CASE nPhase OF
	0:
		// 初始 Undefined -> Aborted。
		Composite(Ctrl := Ctrl, Context := Context, ServiceId := 10);
		nPhase := 1;
	1:
		Ctrl.PackMLIn.eCommand := E_PackMLCommand.Clear;
		Ctrl.PackMLIn.bCommandChangeRequest := TRUE;
		Composite(Ctrl := Ctrl, Context := Context, ServiceId := 10);
		nPhase := 2;
	2:
		Ctrl.PackMLIn.bCommandChangeRequest := FALSE;
		Composite(Ctrl := Ctrl, Context := Context, ServiceId := 10);
		nPhase := 3;
	3:
		Ctrl.PackMLIn.eCommand := E_PackMLCommand.Reset;
		Ctrl.PackMLIn.bCommandChangeRequest := TRUE;
		Composite(Ctrl := Ctrl, Context := Context, ServiceId := 10);
		nPhase := 4;
	4:
		Ctrl.PackMLIn.bCommandChangeRequest := FALSE;
		Composite(Ctrl := Ctrl, Context := Context, ServiceId := 10);
		nPhase := 5;
	5:
		// Starting 發現 definition 尚未設定，加入 framework error 並排入 Stop。
		Ctrl.PackMLIn.eCommand := E_PackMLCommand.Start;
		Ctrl.PackMLIn.bCommandChangeRequest := TRUE;
		Composite(Ctrl := Ctrl, Context := Context, ServiceId := 10);
		AssertTrue(
			Condition :=
				Composite.Status.ErrorList[1].MainErrorId =
				TO_UDINT(E_CompositeServiceErrorCode.NotConfigured),
			Message := 'Unconfigured Composite must publish NotConfigured.'
		);
		nPhase := 6;
	6:
		// 下一掃描由 queued Stop 將 Starting 安全帶回 Stopped。
		Composite(Ctrl := Ctrl, Context := Context, ServiceId := 10);
		AssertTrue(
			Condition := Composite.Status.PackMLOut.eStateCurrent = E_PackMLState.Stopped,
			Message := 'Unconfigured Composite must follow the safe Stop path.'
		);
		nPhase := 0;
		TEST_FINISHED();
END_CASE
END_METHOD

END_FUNCTION_BLOCK

// ---- Fakes/FB_TestCompositeService.TcPOU
FUNCTION_BLOCK FB_TestCompositeService EXTENDS FB_CompositeServiceBase
VAR_INPUT
	DependencyOne : UDINT;
	DependencyTwo : UDINT;
	DependencyCount : UINT;
	ExecuteResult : E_PackMLHookResult := E_PackMLHookResult.Busy;
END_VAR

M_UpdateCompositeService();

METHOD PROTECTED H_DeclareServices
IF DependencyCount >= 1 THEN
	M_AddDependency(ServiceId := DependencyOne);
END_IF
IF DependencyCount >= 2 THEN
	M_AddDependency(ServiceId := DependencyTwo);
END_IF
END_METHOD

METHOD PROTECTED H_OnCompositeExecute : E_PackMLHookResult
VAR_INPUT
	bFirstScan : BOOL;
END_VAR
H_OnCompositeExecute := ExecuteResult;
END_METHOD

METHOD PUBLIC M_TestAddDependencyOutsideDefinition : BOOL
VAR_INPUT
	ServiceIdValue : UDINT;
END_VAR
M_TestAddDependencyOutsideDefinition := M_AddDependency(ServiceId := ServiceIdValue);
END_METHOD

METHOD PUBLIC M_TestFailSequence
VAR_INPUT
	FailedServiceId : UDINT;
END_VAR
M_FailSequence(
	ErrorCode := E_CompositeServiceErrorCode.None,
	FailedServiceId := FailedServiceId,
	SourceErrorId := 0,
	Message := 'Test failure'
);
END_METHOD

END_FUNCTION_BLOCK

// ---- POUs/Test Suites/Service/FB_SetMaterialServiceTests.TcPOU
FUNCTION_BLOCK FB_SetMaterialServiceTests EXTENDS TcUnit.FB_TestSuite

ModifyUsesTheStartingSnapshot();
ClearAndClearAllAffectOnlyTheirDocumentedScope();
InvalidTargetStopsWithAStableError();
MissingTargetIsRejected();
DuplicateTargetIsRejected();
UnsupportedCommandIsRejected();

METHOD ClearAndClearAllAffectOnlyTheirDocumentedScope
VAR_INST
	Service : FB_SetMaterialService;
	Ctrl : ST_ServiceCtrl;
	Context : ST_ServiceContext;
	Param : ST_MaterialParam;
	Wafers : ARRAY[1..2] OF ST_WaferStatus;
	nPhase : UINT;
END_VAR
TEST('ClearAndClearAllAffectOnlyTheirDocumentedScope');

CASE nPhase OF
	0:
		Wafers[1].EndpointId := 1;
		Wafers[2].EndpointId := 2;
		Wafers[1].MaterialContext.Id := 'A';
		Wafers[2].MaterialContext.Id := 'B';
		Service(
			Ctrl := Ctrl,
			Context := Context,
			ServiceId := 2,
			Param := Param,
			WaferStatusList := Wafers
		);
		nPhase := 1;
		1: Ctrl.PackMLIn.eCommand := E_PackMLCommand.Clear;
		Ctrl.PackMLIn.bCommandChangeRequest := TRUE;
		Service(
			Ctrl := Ctrl,
			Context := Context,
			ServiceId := 2,
			Param := Param,
			WaferStatusList := Wafers
		);
		nPhase := 2;
		2: Ctrl.PackMLIn.bCommandChangeRequest := FALSE;
		Service(
			Ctrl := Ctrl,
			Context := Context,
			ServiceId := 2,
			Param := Param,
			WaferStatusList := Wafers
		);
		nPhase := 3;
		3: Ctrl.PackMLIn.eCommand := E_PackMLCommand.Reset;
		Ctrl.PackMLIn.bCommandChangeRequest := TRUE;
		Service(
			Ctrl := Ctrl,
			Context := Context,
			ServiceId := 2,
			Param := Param,
			WaferStatusList := Wafers
		);
		nPhase := 4;
		4: Ctrl.PackMLIn.bCommandChangeRequest := FALSE;
		Service(
			Ctrl := Ctrl,
			Context := Context,
			ServiceId := 2,
			Param := Param,
			WaferStatusList := Wafers
		);
		nPhase := 5;
	5:
		Param.CmdType := E_SetMaterialCmdType.Clear;
		Param.TargetEndpointId := 1;
		Ctrl.PackMLIn.eCommand := E_PackMLCommand.Start;
		Ctrl.PackMLIn.bCommandChangeRequest := TRUE;
		Service(
			Ctrl := Ctrl,
			Context := Context,
			ServiceId := 2,
			Param := Param,
			WaferStatusList := Wafers
		);
		nPhase := 6;
	6:
		Service(
			Ctrl := Ctrl,
			Context := Context,
			ServiceId := 2,
			Param := Param,
			WaferStatusList := Wafers
		);
		AssertTrue(
			Condition := (Wafers[1].MaterialContext.Id = '')
				AND (Wafers[2].MaterialContext.Id = 'B'),
			Message := 'Clear must affect only the selected endpoint.'
		);
		nPhase := 7;
	7:
		Ctrl.PackMLIn.bCommandChangeRequest := FALSE;
		Service(
			Ctrl := Ctrl,
			Context := Context,
			ServiceId := 2,
			Param := Param,
			WaferStatusList := Wafers
		);
		nPhase := 8;
	8:
		Ctrl.PackMLIn.eCommand := E_PackMLCommand.Reset;
		Ctrl.PackMLIn.bCommandChangeRequest := TRUE;
		Service(
			Ctrl := Ctrl,
			Context := Context,
			ServiceId := 2,
			Param := Param,
			WaferStatusList := Wafers
		);
		nPhase := 9;
	9:
		Ctrl.PackMLIn.bCommandChangeRequest := FALSE;
		Service(
			Ctrl := Ctrl,
			Context := Context,
			ServiceId := 2,
			Param := Param,
			WaferStatusList := Wafers
		);
		nPhase := 10;
	10:
		Wafers[1].MaterialContext.Id := 'A2';
		Param.CmdType := E_SetMaterialCmdType.ClearAll;
		Param.TargetEndpointId := 0;
		Ctrl.PackMLIn.eCommand := E_PackMLCommand.Start;
		Ctrl.PackMLIn.bCommandChangeRequest := TRUE;
		Service(
			Ctrl := Ctrl,
			Context := Context,
			ServiceId := 2,
			Param := Param,
			WaferStatusList := Wafers
		);
		nPhase := 11;
	11:
		Service(
			Ctrl := Ctrl,
			Context := Context,
			ServiceId := 2,
			Param := Param,
			WaferStatusList := Wafers
		);
		AssertTrue(
			Condition := (Wafers[1].MaterialContext.Id = '')
				AND (Wafers[2].MaterialContext.Id = ''),
			Message := 'ClearAll must clear every material context and ignore TargetEndpointId.'
		);
		nPhase := 0;
		TEST_FINISHED();
END_CASE
END_METHOD

METHOD DuplicateTargetIsRejected
VAR_INST
	Service : FB_SetMaterialService;
	Ctrl : ST_ServiceCtrl;
	Context : ST_ServiceContext;
	Param : ST_MaterialParam;
	Wafers : ARRAY[1..2] OF ST_WaferStatus;
	nPhase : UINT;
END_VAR
TEST('DuplicateTargetIsRejected');

CASE nPhase OF
	0: Wafers[1].EndpointId := 7;
	Wafers[2].EndpointId := 7;
	Service(
		Ctrl := Ctrl,
		Context := Context,
		ServiceId := 5,
		Param := Param,
		WaferStatusList := Wafers
	);
	nPhase := 1;
	1: Ctrl.PackMLIn.eCommand := E_PackMLCommand.Clear;
	Ctrl.PackMLIn.bCommandChangeRequest := TRUE;
	Service(
		Ctrl := Ctrl,
		Context := Context,
		ServiceId := 5,
		Param := Param,
		WaferStatusList := Wafers
	);
	nPhase := 2;
	2: Ctrl.PackMLIn.bCommandChangeRequest := FALSE;
	Service(
		Ctrl := Ctrl,
		Context := Context,
		ServiceId := 5,
		Param := Param,
		WaferStatusList := Wafers
	);
	nPhase := 3;
	3: Ctrl.PackMLIn.eCommand := E_PackMLCommand.Reset;
	Ctrl.PackMLIn.bCommandChangeRequest := TRUE;
	Service(
		Ctrl := Ctrl,
		Context := Context,
		ServiceId := 5,
		Param := Param,
		WaferStatusList := Wafers
	);
	nPhase := 4;
	4: Ctrl.PackMLIn.bCommandChangeRequest := FALSE;
	Service(
		Ctrl := Ctrl,
		Context := Context,
		ServiceId := 5,
		Param := Param,
		WaferStatusList := Wafers
	);
	nPhase := 5;
	5:
		// Arrange：兩個 storage slot 宣告同一個外部 EndpointId。
		Param.CmdType := E_SetMaterialCmdType.Modify;
		Param.TargetEndpointId := 7;
		Ctrl.PackMLIn.eCommand := E_PackMLCommand.Start;
		Ctrl.PackMLIn.bCommandChangeRequest := TRUE;
		// Act
		Service(
			Ctrl := Ctrl,
			Context := Context,
			ServiceId := 5,
			Param := Param,
			WaferStatusList := Wafers
		);
		// Assert
		AssertTrue(
			Condition :=
				Service.Status.ErrorList[1].MainErrorId =
				TO_UDINT(E_FrameworkServiceErrorCode.SetMaterial_DuplicateTaEpId),
			Message := 'Duplicate target identity must be rejected before modifying either wafer.'
		);
		AssertTrue(
			Condition := (Wafers[1].MaterialContext.Id = '')
				AND (Wafers[2].MaterialContext.Id = ''),
			Message := 'Rejected duplicate target must not mutate material state.'
		);
		nPhase := 0;
		TEST_FINISHED();
END_CASE
END_METHOD

METHOD InvalidTargetStopsWithAStableError
VAR_INST
	Service : FB_SetMaterialService;
	Ctrl : ST_ServiceCtrl;
	Context : ST_ServiceContext;
	Param : ST_MaterialParam;
	Wafers : ARRAY[1..2] OF ST_WaferStatus;
	nPhase : UINT;
END_VAR
TEST('InvalidTargetStopsWithAStableError');

CASE nPhase OF
	0:
		Service(
			Ctrl := Ctrl,
			Context := Context,
			ServiceId := 3,
			Param := Param,
			WaferStatusList := Wafers
		);
		nPhase := 1;
		1: Ctrl.PackMLIn.eCommand := E_PackMLCommand.Clear;
		Ctrl.PackMLIn.bCommandChangeRequest := TRUE;
		Service(
			Ctrl := Ctrl,
			Context := Context,
			ServiceId := 3,
			Param := Param,
			WaferStatusList := Wafers
		);
		nPhase := 2;
		2: Ctrl.PackMLIn.bCommandChangeRequest := FALSE;
		Service(
			Ctrl := Ctrl,
			Context := Context,
			ServiceId := 3,
			Param := Param,
			WaferStatusList := Wafers
		);
		nPhase := 3;
		3: Ctrl.PackMLIn.eCommand := E_PackMLCommand.Reset;
		Ctrl.PackMLIn.bCommandChangeRequest := TRUE;
		Service(
			Ctrl := Ctrl,
			Context := Context,
			ServiceId := 3,
			Param := Param,
			WaferStatusList := Wafers
		);
		nPhase := 4;
		4: Ctrl.PackMLIn.bCommandChangeRequest := FALSE;
		Service(
			Ctrl := Ctrl,
			Context := Context,
			ServiceId := 3,
			Param := Param,
			WaferStatusList := Wafers
		);
		nPhase := 5;
	5:
		// Arrange：Modify/Clear 的 TargetEndpointId=0 是明確輸入錯誤。
		Param.CmdType := E_SetMaterialCmdType.Modify;
		Param.TargetEndpointId := 0;
		Ctrl.PackMLIn.eCommand := E_PackMLCommand.Start;
		Ctrl.PackMLIn.bCommandChangeRequest := TRUE;
		Service(
			Ctrl := Ctrl,
			Context := Context,
			ServiceId := 3,
			Param := Param,
			WaferStatusList := Wafers
		);
		AssertTrue(
			Condition :=
				Service.Status.ErrorList[1].MainErrorId =
				TO_UDINT(E_FrameworkServiceErrorCode.SetMaterial_TaEpIdRequired),
			Message := 'Zero target must publish the required-target error.'
		);
		nPhase := 6;
	6:
		Service(
			Ctrl := Ctrl,
			Context := Context,
			ServiceId := 3,
			Param := Param,
			WaferStatusList := Wafers
		);
		AssertTrue(
			Condition := Service.Status.PackMLOut.eStateCurrent = E_PackMLState.Stopped,
			Message := 'Invalid material request must follow the safe Stop path.'
		);
		nPhase := 0;
		TEST_FINISHED();
END_CASE
END_METHOD

METHOD MissingTargetIsRejected
VAR_INST
	Service : FB_SetMaterialService;
	Ctrl : ST_ServiceCtrl;
	Context : ST_ServiceContext;
	Param : ST_MaterialParam;
	Wafers : ARRAY[1..2] OF ST_WaferStatus;
	nPhase : UINT;
END_VAR
TEST('MissingTargetIsRejected');

CASE nPhase OF
	0: Wafers[1].EndpointId := 10;
	Wafers[2].EndpointId := 20;
	Service(
		Ctrl := Ctrl,
		Context := Context,
		ServiceId := 4,
		Param := Param,
		WaferStatusList := Wafers
	);
	nPhase := 1;
	1: Ctrl.PackMLIn.eCommand := E_PackMLCommand.Clear;
	Ctrl.PackMLIn.bCommandChangeRequest := TRUE;
	Service(
		Ctrl := Ctrl,
		Context := Context,
		ServiceId := 4,
		Param := Param,
		WaferStatusList := Wafers
	);
	nPhase := 2;
	2: Ctrl.PackMLIn.bCommandChangeRequest := FALSE;
	Service(
		Ctrl := Ctrl,
		Context := Context,
		ServiceId := 4,
		Param := Param,
		WaferStatusList := Wafers
	);
	nPhase := 3;
	3: Ctrl.PackMLIn.eCommand := E_PackMLCommand.Reset;
	Ctrl.PackMLIn.bCommandChangeRequest := TRUE;
	Service(
		Ctrl := Ctrl,
		Context := Context,
		ServiceId := 4,
		Param := Param,
		WaferStatusList := Wafers
	);
	nPhase := 4;
	4: Ctrl.PackMLIn.bCommandChangeRequest := FALSE;
	Service(
		Ctrl := Ctrl,
		Context := Context,
		ServiceId := 4,
		Param := Param,
		WaferStatusList := Wafers
	);
	nPhase := 5;
	5:
		// Arrange：使用非零但不存在的 EndpointId。
		Param.CmdType := E_SetMaterialCmdType.Clear;
		Param.TargetEndpointId := 99;
		Ctrl.PackMLIn.eCommand := E_PackMLCommand.Start;
		Ctrl.PackMLIn.bCommandChangeRequest := TRUE;
		// Act
		Service(
			Ctrl := Ctrl,
			Context := Context,
			ServiceId := 4,
			Param := Param,
			WaferStatusList := Wafers
		);
		// Assert
		AssertTrue(
			Condition :=
				Service.Status.ErrorList[1].MainErrorId =
				TO_UDINT(E_FrameworkServiceErrorCode.SetMaterial_TaEpNotFound),
			Message := 'Unknown target must publish the not-found error.'
		);
		nPhase := 0;
		TEST_FINISHED();
END_CASE
END_METHOD

METHOD ModifyUsesTheStartingSnapshot
VAR_INST
	Service : FB_SetMaterialService;
	Ctrl : ST_ServiceCtrl;
	Context : ST_ServiceContext;
	Param : ST_MaterialParam;
	Wafers : ARRAY[1..2] OF ST_WaferStatus;
	nPhase : UINT;
END_VAR
TEST('ModifyUsesTheStartingSnapshot');

CASE nPhase OF
	0:
		Wafers[1].EndpointId := 101;
		Wafers[2].EndpointId := 102;
		Service(
			Ctrl := Ctrl,
			Context := Context,
			ServiceId := 1,
			Param := Param,
			WaferStatusList := Wafers
		);
		nPhase := 1;
	1:
		Ctrl.PackMLIn.eCommand := E_PackMLCommand.Clear;
		Ctrl.PackMLIn.bCommandChangeRequest := TRUE;
		Service(
			Ctrl := Ctrl,
			Context := Context,
			ServiceId := 1,
			Param := Param,
			WaferStatusList := Wafers
		);
		nPhase := 2;
	2:
		Ctrl.PackMLIn.bCommandChangeRequest := FALSE;
		Service(
			Ctrl := Ctrl,
			Context := Context,
			ServiceId := 1,
			Param := Param,
			WaferStatusList := Wafers
		);
		nPhase := 3;
	3:
		Ctrl.PackMLIn.eCommand := E_PackMLCommand.Reset;
		Ctrl.PackMLIn.bCommandChangeRequest := TRUE;
		Service(
			Ctrl := Ctrl,
			Context := Context,
			ServiceId := 1,
			Param := Param,
			WaferStatusList := Wafers
		);
		nPhase := 4;
	4:
		Ctrl.PackMLIn.bCommandChangeRequest := FALSE;
		Service(
			Ctrl := Ctrl,
			Context := Context,
			ServiceId := 1,
			Param := Param,
			WaferStatusList := Wafers
		);
		nPhase := 5;
	5:
		// Arrange：Starting 驗證並 snapshot Modify 參數。
		Param.CmdType := E_SetMaterialCmdType.Modify;
		Param.TargetEndpointId := 101;
		Param.MaterialId := 'WAFER-A';
		Param.MaterialOperateState := E_MaterialOperateState.Processing;
		Ctrl.PackMLIn.eCommand := E_PackMLCommand.Start;
		Ctrl.PackMLIn.bCommandChangeRequest := TRUE;
		Service(
			Ctrl := Ctrl,
			Context := Context,
			ServiceId := 1,
			Param := Param,
			WaferStatusList := Wafers
		);
		Param.MaterialId := 'MUTATED-AFTER-START';
		nPhase := 6;
	6:
		// Act：Execute 必須使用 Starting 的 snapshot，而不是目前輸入。
		Service(
			Ctrl := Ctrl,
			Context := Context,
			ServiceId := 1,
			Param := Param,
			WaferStatusList := Wafers
		);
		AssertTrue(
			Condition :=
				(Wafers[1].MaterialContext.Id = 'WAFER-A')
				AND (Wafers[1].MaterialContext.OperationState = E_MaterialOperateState.Processing),
			Message := 'Modify must use the snapshotted material context.'
		);
		AssertTrue(
			Condition := Wafers[2].MaterialContext.Id = '',
			Message := 'Modify must not change another endpoint.'
		);
		nPhase := 0;
		TEST_FINISHED();
END_CASE
END_METHOD

METHOD UnsupportedCommandIsRejected
VAR_INST
	Service : FB_SetMaterialService;
	Ctrl : ST_ServiceCtrl;
	Context : ST_ServiceContext;
	Param : ST_MaterialParam;
	Wafers : ARRAY[1..2] OF ST_WaferStatus;
	nPhase : UINT;
END_VAR
VAR
	nInvalidCommand : INT := 9999;
END_VAR
TEST('UnsupportedCommandIsRejected');

CASE nPhase OF
	0: Wafers[1].EndpointId := 1;
	Service(
		Ctrl := Ctrl,
		Context := Context,
		ServiceId := 6,
		Param := Param,
		WaferStatusList := Wafers
	);
	nPhase := 1;
	1: Ctrl.PackMLIn.eCommand := E_PackMLCommand.Clear;
	Ctrl.PackMLIn.bCommandChangeRequest := TRUE;
	Service(
		Ctrl := Ctrl,
		Context := Context,
		ServiceId := 6,
		Param := Param,
		WaferStatusList := Wafers
	);
	nPhase := 2;
	2: Ctrl.PackMLIn.bCommandChangeRequest := FALSE;
	Service(
		Ctrl := Ctrl,
		Context := Context,
		ServiceId := 6,
		Param := Param,
		WaferStatusList := Wafers
	);
	nPhase := 3;
	3: Ctrl.PackMLIn.eCommand := E_PackMLCommand.Reset;
	Ctrl.PackMLIn.bCommandChangeRequest := TRUE;
	Service(
		Ctrl := Ctrl,
		Context := Context,
		ServiceId := 6,
		Param := Param,
		WaferStatusList := Wafers
	);
	nPhase := 4;
	4: Ctrl.PackMLIn.bCommandChangeRequest := FALSE;
	Service(
		Ctrl := Ctrl,
		Context := Context,
		ServiceId := 6,
		Param := Param,
		WaferStatusList := Wafers
	);
	nPhase := 5;
	5:
		// Arrange：模擬反序列化或上游資料損壞造成的未知 enum 值。
		// 故意繞過 strict enum 的編譯期保護，模擬外部資料或記憶體損壞。
		MEMCPY(
			ADR(Param.CmdType),
			ADR(nInvalidCommand),
			SIZEOF(Param.CmdType));
		Param.TargetEndpointId := 1;
		Ctrl.PackMLIn.eCommand := E_PackMLCommand.Start;
		Ctrl.PackMLIn.bCommandChangeRequest := TRUE;
		// Act
		Service(
			Ctrl := Ctrl,
			Context := Context,
			ServiceId := 6,
			Param := Param,
			WaferStatusList := Wafers
		);
		// Assert
		AssertTrue(
			Condition :=
				Service.Status.ErrorList[1].MainErrorId =
				TO_UDINT(E_FrameworkServiceErrorCode.SetMaterial_InvalidCmd),
			Message := 'Unknown material command must publish the invalid-command error.'
		);
		nPhase := 0;
		TEST_FINISHED();
END_CASE
END_METHOD

END_FUNCTION_BLOCK

// ---- POUs/Test Suites/Service/FB_ServiceCallerTests.TcPOU
FUNCTION_BLOCK FB_ServiceCallerTests EXTENDS TcUnit.FB_TestSuite

UnconfiguredCallerRejectsRequests();
ConfiguredCallerDelegatesAndAdvancesRequestIds();

METHOD UnconfiguredCallerRejectsRequests
VAR_INST
	Caller : FB_ServiceCaller;
	Param : ST_TestServiceParam;
	Snapshot : ST_ServiceExecutionSnapshot;
END_VAR
TEST('UnconfiguredCallerRejectsRequests');

AssertTrue(
	Condition := Caller.M_Start(
		ServiceId := 1,
		Parameters := Param
	) = E_ServiceCallSubmitResult.CallerNotConfigured,
	Message := 'Unconfigured Start must be rejected.'
);
AssertTrue(
	Condition := Caller.M_Command(
		ServiceId := 1,
		Command := E_PackMLCommand.Stop
	) = E_ServiceCallSubmitResult.CallerNotConfigured,
	Message := 'Unconfigured command must be rejected.'
);
AssertFalse(
	Condition := Caller.M_GetServiceSnapshot(ServiceId := 1, Snapshot => Snapshot),
	Message := 'Unconfigured snapshot query must fail.'
);

TEST_FINISHED();
END_METHOD

METHOD ConfiguredCallerDelegatesAndAdvancesRequestIds
VAR_INST
	Caller : FB_ServiceCaller;
	Coordinator : FB_ServiceCoordinator;
	CompositeUpperCtrl : ST_ServiceCtrl;
	CompositeEffectiveCtrl : ST_ServiceCtrl;
	CompositeUpperParam : ST_TestServiceParam;
	CompositeEffectiveParam : ST_TestServiceParam;
	CompositeStatus : ST_ServiceStatus;
	ChildUpperCtrl : ST_ServiceCtrl;
	ChildEffectiveCtrl : ST_ServiceCtrl;
	ChildUpperParam : ST_TestServiceParam;
	ChildEffectiveParam : ST_TestServiceParam;
	ChildStatus : ST_ServiceStatus;
	ModuleCtrl : ST_ModuleCtrl;
	Dependencies : ARRAY[1..Param_Config.MaxCompositeDependencies] OF UDINT;
	Param : ST_TestServiceParam;
	bInitialized : BOOL;
END_VAR
VAR
	Snapshot : ST_ServiceExecutionSnapshot;
END_VAR
TEST('ConfiguredCallerDelegatesAndAdvancesRequestIds');

IF NOT bInitialized THEN
	Coordinator.M_BeginRegistration();
	Coordinator.M_Register(
		ServiceId := 10,
		AllowCompositeCall := FALSE,
		UpperCtrl := CompositeUpperCtrl,
		EffectiveCtrl := CompositeEffectiveCtrl,
		UpperParam := CompositeUpperParam,
		EffectiveParam := CompositeEffectiveParam,
		Status := CompositeStatus
	);
	Coordinator.M_Register(
		ServiceId := 20,
		AllowCompositeCall := TRUE,
		UpperCtrl := ChildUpperCtrl,
		EffectiveCtrl := ChildEffectiveCtrl,
		UpperParam := ChildUpperParam,
		EffectiveParam := ChildEffectiveParam,
		Status := ChildStatus
	);
	Dependencies[1] := 20;
	Coordinator.M_RegisterCompositeDefinition(
		CompositeServiceId := 10,
		DependencyCount := 1,
		DependencyIds := Dependencies
	);
	Coordinator.M_Seal();
	ChildStatus.PackMLOut.eStateCurrent := E_PackMLState.Idle;
	ChildStatus.CompletionBehavior := E_ServiceCompletionBehavior.NaturalCompletion;
	Coordinator.M_ObserveCycle();
	Coordinator.M_RequestCompositeOwnership(CompositeServiceId := 10);
	Coordinator.M_PrepareCycle(ModuleInExecute := TRUE, ModuleCtrl := ModuleCtrl);
	AssertTrue(
		Condition := Caller.M_Configure(CallerServiceId := 10, Coordinator := Coordinator),
		Message := 'Registered Composite caller must configure.'
	);
	bInitialized := TRUE;
END_IF

Param.Value := 7;
Param.Sequence := 8;
AssertTrue(
	Condition := Caller.M_Start(
		ServiceId := 20,
		Parameters := Param
	) = E_ServiceCallSubmitResult.Queued,
	Message := 'Caller must delegate Start.'
);
Coordinator.M_PrepareCycle(ModuleInExecute := TRUE, ModuleCtrl := ModuleCtrl);
AssertTrue(
	Condition := ChildEffectiveCtrl.RequestId = 1,
	Message := 'First successful caller request ID must be one.'
);
ChildStatus.ResponseId := 1;
ChildStatus.PackMLOut.bCommandAccepted := TRUE;
Coordinator.M_ObserveCycle();
AssertTrue(
	Condition := Caller.M_GetCommandState(ServiceId := 20) =
		E_ServiceInternalCommandState.Accepted,
	Message := 'Caller must expose Coordinator command state.'
);
AssertTrue(
	Condition := Caller.M_GetServiceSnapshot(
		ServiceId := 20,
		Snapshot => Snapshot
	) AND Snapshot.Valid,
	Message := 'Caller must expose the observed Service snapshot.'
);
Coordinator.M_PrepareCycle(ModuleInExecute := TRUE, ModuleCtrl := ModuleCtrl);
// 強制 low 一掃描。
AssertTrue(
	Condition := Caller.M_Command(
		ServiceId := 20,
		Command := E_PackMLCommand.Stop
	) = E_ServiceCallSubmitResult.Queued,
	Message := 'A later lifecycle command must queue.'
);
Coordinator.M_PrepareCycle(ModuleInExecute := TRUE, ModuleCtrl := ModuleCtrl);
AssertTrue(
	Condition := ChildEffectiveCtrl.RequestId = 2,
	Message := 'Only successful queued requests advance the caller ID.'
);

TEST_FINISHED();
END_METHOD

END_FUNCTION_BLOCK

// ---- POUs/Test Suites/Service/FB_ServiceCoordinatorTests.TcPOU
FUNCTION_BLOCK FB_ServiceCoordinatorTests EXTENDS TcUnit.FB_TestSuite

RegistrationRejectsInvalidAndDuplicateServices();
UpperStartSnapshotsParametersOnlyOnNewEdge();
ModuleLifecycleWhitelistAndCompositeHandshakeAreEnforced();

METHOD RegistrationRejectsInvalidAndDuplicateServices
VAR_INST
	Coordinator : FB_ServiceCoordinator;
	UpperCtrl : ST_ServiceCtrl;
	EffectiveCtrl : ST_ServiceCtrl;
	UpperParam : ST_TestServiceParam;
	EffectiveParam : ST_TestServiceParam;
	Status : ST_ServiceStatus;
END_VAR
TEST('RegistrationRejectsInvalidAndDuplicateServices');

// Arrange：先開始一次 registration session。
AssertTrue(
	Condition := Coordinator.M_BeginRegistration(),
	Message := 'Registration must begin exactly once.'
);

// Act / Assert：ServiceId=0 是第一個錯誤，後續註冊不得覆蓋。
AssertFalse(
	Condition := Coordinator.M_Register(
		ServiceId := 0,
		AllowCompositeCall := FALSE,
		UpperCtrl := UpperCtrl,
		EffectiveCtrl := EffectiveCtrl,
		UpperParam := UpperParam,
		EffectiveParam := EffectiveParam,
		Status := Status
	),
	Message := 'ServiceId zero must be rejected.'
);
AssertTrue(
	Condition := Coordinator.RegistrationError = E_ServiceRegistrationError.InvalidServiceId,
	Message := 'Invalid ServiceId must expose a stable error.'
);
AssertFalse(
	Condition := Coordinator.M_Register(
		ServiceId := 1,
		AllowCompositeCall := FALSE,
		UpperCtrl := UpperCtrl,
		EffectiveCtrl := EffectiveCtrl,
		UpperParam := UpperParam,
		EffectiveParam := EffectiveParam,
		Status := Status
	),
	Message := 'A latched registration error must block later writes.'
);
AssertTrue(
	Condition := Coordinator.FailedServiceId = 0,
	Message := 'First-error identity must be preserved.'
);

TEST_FINISHED();
END_METHOD

METHOD UpperStartSnapshotsParametersOnlyOnNewEdge
VAR_INST
	Coordinator : FB_ServiceCoordinator;
	UpperCtrl : ST_ServiceCtrl;
	EffectiveCtrl : ST_ServiceCtrl;
	UpperParam : ST_TestServiceParam;
	EffectiveParam : ST_TestServiceParam;
	Status : ST_ServiceStatus;
	ModuleCtrl : ST_ModuleCtrl;
	bInitialized : BOOL;
END_VAR
TEST('UpperStartSnapshotsParametersOnlyOnNewEdge');

IF NOT bInitialized THEN
	// Arrange：以 suite instance 儲存區註冊，確保 reflection 可取得真實 DUT 名稱。
	Coordinator.M_BeginRegistration();
	AssertTrue(
		Condition := Coordinator.M_Register(
			ServiceId := 1,
			AllowCompositeCall := FALSE,
			UpperCtrl := UpperCtrl,
			EffectiveCtrl := EffectiveCtrl,
			UpperParam := UpperParam,
			EffectiveParam := EffectiveParam,
			Status := Status
		),
		Message := 'Valid Service storage must register.'
	);
	AssertTrue(
		Condition := Coordinator.M_Seal(),
		Message := 'A non-empty valid registry must seal.'
	);
	bInitialized := TRUE;
END_IF

// Act：新的 Start 上升沿 snapshot UpperParam。
UpperParam.Value := 10;
UpperParam.Sequence := 1;
UpperCtrl.RequestId := 100;
UpperCtrl.PackMLIn.eCommand := E_PackMLCommand.Start;
UpperCtrl.PackMLIn.bCommandChangeRequest := TRUE;
Coordinator.M_PrepareCycle(ModuleInExecute := TRUE, ModuleCtrl := ModuleCtrl);
AssertTrue(
	Condition :=
		EffectiveCtrl.PackMLIn.bCommandChangeRequest
		AND (EffectiveParam.Value = 10)
		AND (EffectiveParam.Sequence = 1),
	Message := 'New Start edge must copy control and parameters.'
);

// request 保持高位時，變更 UpperParam 不可污染本次執行 snapshot。
UpperParam.Value := 99;
UpperParam.Sequence := 2;
Coordinator.M_PrepareCycle(ModuleInExecute := TRUE, ModuleCtrl := ModuleCtrl);
AssertTrue(
	Condition := (EffectiveParam.Value = 10) AND (EffectiveParam.Sequence = 1),
	Message := 'Held Start request must keep the first parameter snapshot.'
);

// Falling edge re-arm，下一個 Start 才能取得新參數。
UpperCtrl.PackMLIn.bCommandChangeRequest := FALSE;
Coordinator.M_PrepareCycle(ModuleInExecute := TRUE, ModuleCtrl := ModuleCtrl);
UpperCtrl.PackMLIn.bCommandChangeRequest := TRUE;
Coordinator.M_PrepareCycle(ModuleInExecute := TRUE, ModuleCtrl := ModuleCtrl);
AssertTrue(
	Condition := (EffectiveParam.Value = 99) AND (EffectiveParam.Sequence = 2),
	Message := 'A new Start edge must refresh the snapshot.'
);

TEST_FINISHED();
END_METHOD

METHOD ModuleLifecycleWhitelistAndCompositeHandshakeAreEnforced
VAR_INST
	Coordinator : FB_ServiceCoordinator;
	CompositeUpperCtrl : ST_ServiceCtrl;
	CompositeEffectiveCtrl : ST_ServiceCtrl;
	CompositeUpperParam : ST_TestServiceParam;
	CompositeEffectiveParam : ST_TestServiceParam;
	CompositeStatus : ST_ServiceStatus;
	ChildUpperCtrl : ST_ServiceCtrl;
	ChildEffectiveCtrl : ST_ServiceCtrl;
	ChildUpperParam : ST_TestServiceParam;
	ChildEffectiveParam : ST_TestServiceParam;
	ChildStatus : ST_ServiceStatus;
	ModuleCtrl : ST_ModuleCtrl;
	Dependencies : ARRAY[1..Param_Config.MaxCompositeDependencies] OF UDINT;
	StartParam : ST_TestServiceParam;
	bInitialized : BOOL;
END_VAR
VAR
	Submit : E_ServiceCallSubmitResult;
	Ownership : E_CompositeOwnershipState;
END_VAR
TEST('ModuleLifecycleWhitelistAndCompositeHandshakeAreEnforced');

IF NOT bInitialized THEN
	Coordinator.M_BeginRegistration();
	Coordinator.M_Register(
		ServiceId := 10,
		AllowCompositeCall := FALSE,
		UpperCtrl := CompositeUpperCtrl,
		EffectiveCtrl := CompositeEffectiveCtrl,
		UpperParam := CompositeUpperParam,
		EffectiveParam := CompositeEffectiveParam,
		Status := CompositeStatus
	);
	Coordinator.M_Register(
		ServiceId := 20,
		AllowCompositeCall := TRUE,
		UpperCtrl := ChildUpperCtrl,
		EffectiveCtrl := ChildEffectiveCtrl,
		UpperParam := ChildUpperParam,
		EffectiveParam := ChildEffectiveParam,
		Status := ChildStatus
	);
	Dependencies[1] := 20;
	AssertTrue(
		Condition := Coordinator.M_RegisterCompositeDefinition(
			CompositeServiceId := 10,
			DependencyCount := 1,
			DependencyIds := Dependencies
		),
		Message := 'Valid Composite definition must register.'
	);
	AssertTrue(
		Condition := Coordinator.M_Seal(),
		Message := 'Composite registry must seal.'
	);
	ChildStatus.PackMLOut.eStateCurrent := E_PackMLState.Idle;
	ChildStatus.CompletionBehavior := E_ServiceCompletionBehavior.NaturalCompletion;
	Coordinator.M_ObserveCycle();
	AssertTrue(
		Condition := Coordinator.M_RequestCompositeOwnership(CompositeServiceId := 10),
		Message := 'Composite ownership request must queue.'
	);
	Coordinator.M_PrepareCycle(ModuleInExecute := TRUE, ModuleCtrl := ModuleCtrl);
	Ownership := Coordinator.M_GetCompositeOwnershipState(CompositeServiceId := 10);
	AssertTrue(
		Condition := Ownership = E_CompositeOwnershipState.Owned,
		Message := 'Idle NaturalCompletion dependency must be owned atomically.'
	);
	bInitialized := TRUE;
END_IF

// Act：內部 Start 排入後，高位維持到 Service 回覆相同 RequestId。
StartParam.Value := 55;
StartParam.Sequence := 9;
Submit := Coordinator.M_SubmitInternalStart(
	CallerServiceId := 10,
	TargetServiceId := 20,
	RequestId := 123,
	Parameters := StartParam
);
AssertTrue(
	Condition := Submit = E_ServiceCallSubmitResult.Queued,
	Message := 'Owner may queue dependency Start.'
);
AssertTrue(
	Condition := Coordinator.M_SubmitInternalCommand(
		CallerServiceId := 10,
		TargetServiceId := 20,
		RequestId := 124,
		Command := E_PackMLCommand.Stop
	) = E_ServiceCallSubmitResult.Busy,
	Message := 'A second internal request must be busy.'
);
Coordinator.M_PrepareCycle(ModuleInExecute := TRUE, ModuleCtrl := ModuleCtrl);
AssertTrue(
	Condition :=
		ChildEffectiveCtrl.PackMLIn.bCommandChangeRequest
		AND (ChildEffectiveCtrl.RequestId = 123)
		AND (ChildEffectiveParam.Value = 55),
	Message := 'Queued Start must become the effective child request.'
);
ChildStatus.ResponseId := 123;
ChildStatus.PackMLOut.bCommandAccepted := TRUE;
Coordinator.M_ObserveCycle();
AssertTrue(
	Condition := Coordinator.M_GetInternalCommandState(
		CallerServiceId := 10,
		TargetServiceId := 20
	) = E_ServiceInternalCommandState.Accepted,
	Message := 'Matching accepted response must finish the handshake.'
);
Coordinator.M_PrepareCycle(ModuleInExecute := TRUE, ModuleCtrl := ModuleCtrl);
AssertFalse(
	Condition := ChildEffectiveCtrl.PackMLIn.bCommandChangeRequest,
	Message := 'Accepted request must be forced low for one scan.'
);

// Module 離開 Execute 時只允許 Stop/Abort/Clear/Reset；Start 必須被清除。
ModuleCtrl.PackMLIn.eCommand := E_PackMLCommand.Start;
ModuleCtrl.PackMLIn.bCommandChangeRequest := TRUE;
Coordinator.M_PrepareCycle(ModuleInExecute := FALSE, ModuleCtrl := ModuleCtrl);
AssertFalse(
	Condition := ChildEffectiveCtrl.PackMLIn.bCommandChangeRequest,
	Message := 'Module Start must never fan out to Services.'
);
ModuleCtrl.PackMLIn.eCommand := E_PackMLCommand.Stop;
Coordinator.M_PrepareCycle(ModuleInExecute := FALSE, ModuleCtrl := ModuleCtrl);
AssertTrue(
	Condition :=
		ChildEffectiveCtrl.PackMLIn.bCommandChangeRequest
		AND (ChildEffectiveCtrl.PackMLIn.eCommand = E_PackMLCommand.Stop),
	Message := 'Module Stop must fan out to Services.'
);

TEST_FINISHED();
END_METHOD

END_FUNCTION_BLOCK

// ---- POUs/Test Suites/Module/FB_ModuleAlarmManagerTests.TcPOU
FUNCTION_BLOCK FB_ModuleAlarmManagerTests EXTENDS TcUnit.FB_TestSuite
VAR
	_LifecycleManager : FB_ModuleAlarmManager;
	_AckManager : FB_ModuleAlarmManager;
	_ScopeManager : FB_ModuleAlarmManager;
	_OverflowManager : FB_ModuleAlarmManager;
	_ConfiguredManager : FB_ModuleAlarmManager;
	_HookLifecycleManager : FB_ModuleAlarmManager;
	_HookAckManager : FB_ModuleAlarmManager;
	_HookCapacityManager : FB_ModuleAlarmManager;
	_AlarmList : ARRAY[1..Param_Config.MaxPublishedModuleAlarms] OF ST_ExtAlarm;
END_VAR

HookCapacityAndConfigurationOwnershipHaveSeparateResetScopes();
HookAcknowledgementsRespectIdentityAndNewEventOrdering();
HookOccurrencesUseTheExistingAcknowledgementLifecycle();
ServiceOccurrenceCountChangesOnlyOnActiveEdges();
AcknowledgeOneUsesCompositeIdentityAndRemovalPredicate();
AcknowledgementPrecedesNewSourcesAndResetsHaveSeparateScopes();
ConfiguredOccurrencesAndDuplicateRequestsFollowTheSameContract();
ServiceOverflowPreservesExistingLifecycles();

METHOD ServiceOccurrenceCountChangesOnlyOnActiveEdges
VAR
	Alarm : ST_ExtAlarm;
END_VAR
TEST('ServiceOccurrenceCountChangesOnlyOnActiveEdges');

Alarm.ModuleId := 1;
Alarm.ServiceId := 11;
Alarm.MainErrorId := 101;
Alarm.SourceErrorId := 16#1234;
Alarm.Message := 'First occurrence';
Alarm.Path := 'Chamber1.Service11';
Alarm.Severity := E_Severity.Alarm;
Alarm.DateTime := '20260828090000000';

// First rising edge creates the lifecycle with count 1.
_LifecycleManager.M_BeginCycle(ModuleId := 1, ConfigurationRevision := 1);
_LifecycleManager.M_ObserveServiceAlarm(Alarm := Alarm);
_LifecycleManager.M_EndCycle();
_LifecycleManager.M_Publish(AlarmList := _AlarmList);
AssertTrue(
	Condition := _AlarmList[1].Active,
	Message := 'First observation must publish an active alarm.'
);
AssertTrue(
	Condition := _AlarmList[1].OccurrenceCount = 1,
	Message := 'First active edge must set occurrence count to one.'
);

// Continuous presence is not another active edge.
_LifecycleManager.M_BeginCycle(ModuleId := 1, ConfigurationRevision := 1);
_LifecycleManager.M_ObserveServiceAlarm(Alarm := Alarm);
_LifecycleManager.M_EndCycle();
_LifecycleManager.M_Publish(AlarmList := _AlarmList);
AssertTrue(
	Condition := _AlarmList[1].OccurrenceCount = 1,
	Message := 'Continuous active scans must not increase occurrence count.'
);

// Absence makes the retained lifecycle inactive.
_LifecycleManager.M_BeginCycle(ModuleId := 1, ConfigurationRevision := 1);
_LifecycleManager.M_EndCycle();
_LifecycleManager.M_Publish(AlarmList := _AlarmList);
AssertFalse(
	Condition := _AlarmList[1].Active,
	Message := 'A missing Service source must make the retained alarm inactive.'
);

// Reappearance before acknowledgement is a second active edge.
// The first occurrence metadata remains latched.
Alarm.SourceErrorId := 16#5678;
Alarm.Message := 'Later occurrence';
Alarm.DateTime := '20260828090100000';
_LifecycleManager.M_BeginCycle(ModuleId := 1, ConfigurationRevision := 1);
_LifecycleManager.M_ObserveServiceAlarm(Alarm := Alarm);
_LifecycleManager.M_EndCycle();
_LifecycleManager.M_Publish(AlarmList := _AlarmList);
AssertTrue(
	Condition := _AlarmList[1].Active,
	Message := 'A recurring source must become active again.'
);
AssertTrue(
	Condition := _AlarmList[1].OccurrenceCount = 2,
	Message := 'Only the recurring active edge may increase occurrence count.'
);
AssertFalse(
	Condition := _AlarmList[1].Acknowledged,
	Message := 'A recurrence must require acknowledgement again.'
);
AssertTrue(
	Condition := _AlarmList[1].SourceErrorId = 16#1234,
	Message := 'A recurrence must retain the first source error ID.'
);
AssertTrue(
	Condition := _AlarmList[1].Message = 'First occurrence',
	Message := 'A recurrence must retain the first message.'
);
AssertTrue(
	Condition := _AlarmList[1].DateTime = '20260828090000000',
	Message := 'A recurrence must retain the first timestamp.'
);

TEST_FINISHED();
END_METHOD

METHOD AcknowledgeOneUsesCompositeIdentityAndRemovalPredicate
VAR
	AlarmOne : ST_ExtAlarm;
	AlarmTwo : ST_ExtAlarm;
	Request : ST_AlarmAckRequest;
END_VAR
TEST('AcknowledgeOneUsesCompositeIdentityAndRemovalPredicate');

AlarmOne.ModuleId := 2;
AlarmOne.ServiceId := 21;
AlarmOne.MainErrorId := 500;
AlarmOne.Message := 'Service 21';
AlarmOne.DateTime := '20260828100000000';
AlarmTwo := AlarmOne;
AlarmTwo.ServiceId := 22;
AlarmTwo.Message := 'Service 22';

_AckManager.M_BeginCycle(ModuleId := 2, ConfigurationRevision := 1);
_AckManager.M_ObserveServiceAlarm(Alarm := AlarmOne);
_AckManager.M_ObserveServiceAlarm(Alarm := AlarmTwo);
_AckManager.M_EndCycle();

Request.RequestId := 1;
Request.Command := E_AlarmAckCommand.AcknowledgeOne;
Request.MainErrorId := 500;
Request.bChangeRequest := TRUE;
Request.ServiceId := 21;
_AckManager.M_BeginCycle(ModuleId := 2, ConfigurationRevision := 1);
_AckManager.M_ProcessAcknowledgement(Request := Request);
_AckManager.M_ObserveServiceAlarm(Alarm := AlarmOne);
_AckManager.M_ObserveServiceAlarm(Alarm := AlarmTwo);
_AckManager.M_EndCycle();
_AckManager.M_Publish(AlarmList := _AlarmList);
AssertTrue(
	Condition := _AckManager.AckAccepted,
	Message := 'A matching composite identity must be acknowledged.'
);
AssertTrue(
	Condition := _AlarmList[1].ServiceId = 21 AND _AlarmList[1].Acknowledged,
	Message := 'Only Service 21 must be acknowledged.'
);
AssertTrue(
	Condition := _AlarmList[2].ServiceId = 22 AND NOT _AlarmList[2].Acknowledged,
	Message := 'The same error ID from Service 22 must remain unacknowledged.'
);

// Release the request and remove only the acknowledged alarm by making it inactive.
Request.bChangeRequest := FALSE;
_AckManager.M_BeginCycle(ModuleId := 2, ConfigurationRevision := 1);
_AckManager.M_ProcessAcknowledgement(Request := Request);
_AckManager.M_ObserveServiceAlarm(Alarm := AlarmTwo);
_AckManager.M_EndCycle();
_AckManager.M_Publish(AlarmList := _AlarmList);
AssertTrue(
	Condition := _AlarmList[1].ServiceId = 22,
	Message := 'Inactive and acknowledged Service 21 must be removed in the same scan.'
);
AssertTrue(
	Condition := _AlarmList[2].MainErrorId = 0,
	Message := 'Published alarms must remain dense after removal.'
);

// Reset-before-Ack retains Service 22 as inactive until its exact identity is acknowledged.
_AckManager.M_BeginCycle(ModuleId := 2, ConfigurationRevision := 1);
_AckManager.M_EndCycle();
_AckManager.M_Publish(AlarmList := _AlarmList);
AssertFalse(
	Condition := _AlarmList[1].Active,
	Message := 'An inactive unacknowledged alarm must remain published.'
);

Request.RequestId := 2;
Request.ServiceId := 22;
Request.bChangeRequest := TRUE;
_AckManager.M_BeginCycle(ModuleId := 2, ConfigurationRevision := 1);
_AckManager.M_ProcessAcknowledgement(Request := Request);
_AckManager.M_EndCycle();
_AckManager.M_Publish(AlarmList := _AlarmList);
AssertTrue(
	Condition := _AlarmList[1].MainErrorId = 0,
	Message := 'Acknowledging an inactive alarm must remove it in the same scan.'
);
AssertTrue(
	Condition := _AckManager.AckResponseId = 2 AND _AckManager.AckAccepted,
	Message := 'Ack response must identify the accepted request.'
);

TEST_FINISHED();
END_METHOD

METHOD AcknowledgementPrecedesNewSourcesAndResetsHaveSeparateScopes
VAR
	ServiceAlarm : ST_ExtAlarm;
	ConfiguredAlarm : ST_ExtAlarm;
	Request : ST_AlarmAckRequest;
END_VAR
TEST('AcknowledgementPrecedesNewSourcesAndResetsHaveSeparateScopes');

ServiceAlarm.ModuleId := 3;
ServiceAlarm.ServiceId := 31;
ServiceAlarm.MainErrorId := 601;
ServiceAlarm.Message := 'Service alarm';
ServiceAlarm.DateTime := '20260828110000000';
ConfiguredAlarm.ModuleId := 3;
ConfiguredAlarm.ServiceId := 99;
ConfiguredAlarm.MainErrorId := 602;
ConfiguredAlarm.Message := 'Configured alarm';
ConfiguredAlarm.Severity := E_Severity.Warning;

// AckAll happens before either new source is sampled, so neither new lifecycle is acknowledged.
Request.RequestId := 10;
Request.Command := E_AlarmAckCommand.AcknowledgeAll;
Request.bChangeRequest := TRUE;
_ScopeManager.M_BeginCycle(ModuleId := 3, ConfigurationRevision := 1);
_ScopeManager.M_ProcessAcknowledgement(Request := Request);
_ScopeManager.M_UpdateConfiguredAlarm(
	AlarmIndex := 1,
	SampleValid := TRUE,
	ConditionMet := TRUE,
	Alarm := ConfiguredAlarm,
	UtcDateTime := '20260828110000000');
_ScopeManager.M_ObserveServiceAlarm(Alarm := ServiceAlarm);
_ScopeManager.M_EndCycle();
_ScopeManager.M_Publish(AlarmList := _AlarmList);
AssertTrue(
	Condition := _AlarmList[1].ServiceId = 31 AND NOT _AlarmList[1].Acknowledged,
	Message := 'AckAll must not consume a new Service alarm from the same scan.'
);
AssertTrue(
	Condition := _AlarmList[2].ServiceId = 0 AND NOT _AlarmList[2].Acknowledged,
	Message := 'Configured alarms must publish with ServiceId zero and require a later Ack.'
);
AssertTrue(
	Condition := _ScopeManager.ServiceLatchedCount = 1,
	Message := 'Service latched count must include the Service lifecycle.'
);
AssertTrue(
	Condition := _ScopeManager.ConfiguredLatchedCount = 1,
	Message := 'Configured latched count must include the configured lifecycle.'
);

// A configuration revision clears only configured state and preserves the Service lifecycle.
Request.bChangeRequest := FALSE;
_ScopeManager.M_BeginCycle(ModuleId := 3, ConfigurationRevision := 2);
_ScopeManager.M_ProcessAcknowledgement(Request := Request);
_ScopeManager.M_ObserveServiceAlarm(Alarm := ServiceAlarm);
_ScopeManager.M_EndCycle();
_ScopeManager.M_Publish(AlarmList := _AlarmList);
AssertTrue(
	Condition := _ScopeManager.ServiceLatchedCount = 1,
	Message := 'Configuration revision changes must preserve Service alarms.'
);
AssertTrue(
	Condition := _ScopeManager.ConfiguredLatchedCount = 0,
	Message := 'Configuration revision changes must clear configured alarms.'
);

// Reassigning the FB instance to another Module identity clears both scopes.
_ScopeManager.M_BeginCycle(ModuleId := 4, ConfigurationRevision := 2);
_ScopeManager.M_EndCycle();
_ScopeManager.M_Publish(AlarmList := _AlarmList);
AssertTrue(
	Condition := _ScopeManager.ServiceLatchedCount = 0
		AND _ScopeManager.ConfiguredLatchedCount = 0,
	Message := 'A ModuleId change must clear every alarm lifecycle.'
);
AssertTrue(
	Condition := _AlarmList[1].MainErrorId = 0,
	Message := 'A ModuleId change must publish an empty list.'
);

TEST_FINISHED();
END_METHOD

METHOD ServiceOverflowPreservesExistingLifecycles
VAR
	Alarm : ST_ExtAlarm;
	nIndex : UINT;
END_VAR
TEST('ServiceOverflowPreservesExistingLifecycles');

_OverflowManager.M_BeginCycle(ModuleId := 5, ConfigurationRevision := 1);
FOR nIndex := 1 TO Param_Config.MaxServiceAlarmsPerModule + 1 DO
	Alarm.ModuleId := 5;
	Alarm.ServiceId := nIndex;
	Alarm.MainErrorId := 1000 + nIndex;
	Alarm.Message := 'Capacity test';
	Alarm.DateTime := '20260828120000000';
	_OverflowManager.M_ObserveServiceAlarm(Alarm := Alarm);
END_FOR
_OverflowManager.M_EndCycle();
_OverflowManager.M_Publish(AlarmList := _AlarmList);

AssertTrue(
	Condition := _OverflowManager.ServiceLatchedCount =
		Param_Config.MaxServiceAlarmsPerModule,
	Message := 'Service alarm storage must stop at its fixed capacity.'
);
AssertTrue(
	Condition := _OverflowManager.Overflow,
	Message := 'Rejecting a new alarm at capacity must set Overflow.'
);
AssertTrue(
	Condition := _AlarmList[Param_Config.MaxServiceAlarmsPerModule].MainErrorId <> 0,
	Message := 'The final available slot must remain published.'
);
AssertTrue(
	Condition := _AlarmList[Param_Config.MaxServiceAlarmsPerModule + 1].MainErrorId = 0,
	Message := 'Overflow must not overwrite or publish beyond the reserved Service capacity.'
);

TEST_FINISHED();
END_METHOD

METHOD ConfiguredOccurrencesAndDuplicateRequestsFollowTheSameContract
VAR
	Alarm : ST_ExtAlarm;
	Request : ST_AlarmAckRequest;
END_VAR
TEST('ConfiguredOccurrencesAndDuplicateRequestsFollowTheSameContract');

Alarm.ModuleId := 6;
Alarm.ServiceId := 999;
Alarm.MainErrorId := 700;
Alarm.SourceErrorId := 701;
Alarm.Message := 'First configured occurrence';
Alarm.Path := 'GVL.Condition';
Alarm.Severity := E_Severity.Alarm;

_ConfiguredManager.M_BeginCycle(ModuleId := 6, ConfigurationRevision := 1);
_ConfiguredManager.M_UpdateConfiguredAlarm(
	AlarmIndex := 1,
	SampleValid := TRUE,
	ConditionMet := TRUE,
	Alarm := Alarm,
	UtcDateTime := '20260828140000000'
);
_ConfiguredManager.M_EndCycle();
_ConfiguredManager.M_Publish(AlarmList := _AlarmList);
AssertTrue(
	Condition := (_AlarmList[1].ServiceId = 0) AND (_AlarmList[1].OccurrenceCount = 1),
	Message := 'Configured alarm first edge must use ServiceId zero and count one.'
);

// Continuous true does not count; false followed by true before removal does.
_ConfiguredManager.M_BeginCycle(ModuleId := 6, ConfigurationRevision := 1);
_ConfiguredManager.M_UpdateConfiguredAlarm(
	AlarmIndex := 1,
	SampleValid := TRUE,
	ConditionMet := TRUE,
	Alarm := Alarm,
	UtcDateTime := '20260828140100000'
);
_ConfiguredManager.M_EndCycle();
_ConfiguredManager.M_Publish(AlarmList := _AlarmList);
AssertTrue(
	Condition := _AlarmList[1].OccurrenceCount = 1,
	Message := 'Continuous configured condition must not increase occurrence count.'
);

_ConfiguredManager.M_BeginCycle(ModuleId := 6, ConfigurationRevision := 1);
_ConfiguredManager.M_UpdateConfiguredAlarm(
	AlarmIndex := 1,
	SampleValid := TRUE,
	ConditionMet := FALSE,
	Alarm := Alarm,
	UtcDateTime := '20260828140200000'
);
_ConfiguredManager.M_EndCycle();
_ConfiguredManager.M_BeginCycle(ModuleId := 6, ConfigurationRevision := 1);
_ConfiguredManager.M_UpdateConfiguredAlarm(
	AlarmIndex := 1,
	SampleValid := TRUE,
	ConditionMet := TRUE,
	Alarm := Alarm,
	UtcDateTime := '20260828140300000'
);
_ConfiguredManager.M_EndCycle();
_ConfiguredManager.M_Publish(AlarmList := _AlarmList);
AssertTrue(
	Condition := _AlarmList[1].OccurrenceCount = 2,
	Message :=
		'Configured recurrence before removal must increment only on the new active edge.'
);
AssertTrue(
	Condition := _AlarmList[1].DateTime = '20260828140000000',
	Message := 'Configured recurrence must retain the first lifecycle timestamp.'
);

Request.RequestId := 20;
Request.Command := E_AlarmAckCommand.AcknowledgeOne;
Request.MainErrorId := 700;
Request.ServiceId := 0;
Request.bChangeRequest := TRUE;
_ConfiguredManager.M_BeginCycle(ModuleId := 6, ConfigurationRevision := 1);
_ConfiguredManager.M_ProcessAcknowledgement(Request := Request);
_ConfiguredManager.M_UpdateConfiguredAlarm(
	AlarmIndex := 1,
	SampleValid := TRUE,
	ConditionMet := TRUE,
	Alarm := Alarm,
	UtcDateTime := '20260828140400000'
);
_ConfiguredManager.M_EndCycle();
AssertTrue(
	Condition := _ConfiguredManager.AckAccepted,
	Message := 'Configured AcknowledgeOne must accept ServiceId zero.'
);

Request.bChangeRequest := FALSE;
_ConfiguredManager.M_BeginCycle(ModuleId := 6, ConfigurationRevision := 1);
_ConfiguredManager.M_ProcessAcknowledgement(Request := Request);
_ConfiguredManager.M_UpdateConfiguredAlarm(
	AlarmIndex := 1,
	SampleValid := TRUE,
	ConditionMet := TRUE,
	Alarm := Alarm,
	UtcDateTime := '20260828140500000'
);
_ConfiguredManager.M_EndCycle();
Request.bChangeRequest := TRUE;
_ConfiguredManager.M_BeginCycle(ModuleId := 6, ConfigurationRevision := 1);
_ConfiguredManager.M_ProcessAcknowledgement(Request := Request);
_ConfiguredManager.M_UpdateConfiguredAlarm(
	AlarmIndex := 1,
	SampleValid := TRUE,
	ConditionMet := TRUE,
	Alarm := Alarm,
	UtcDateTime := '20260828140600000'
);
_ConfiguredManager.M_EndCycle();
AssertTrue(
	Condition := _ConfiguredManager.AckError = E_AlarmAckError.DuplicateRequest,
	Message := 'A repeated nonzero RequestId after a new request edge must be rejected.'
);

// The accepted Ack remains on the active alarm; the later false sample removes it immediately.
Request.bChangeRequest := FALSE;
_ConfiguredManager.M_BeginCycle(ModuleId := 6, ConfigurationRevision := 1);
_ConfiguredManager.M_ProcessAcknowledgement(Request := Request);
_ConfiguredManager.M_UpdateConfiguredAlarm(
	AlarmIndex := 1,
	SampleValid := TRUE,
	ConditionMet := FALSE,
	Alarm := Alarm,
	UtcDateTime := '20260828140700000'
);
_ConfiguredManager.M_EndCycle();
_ConfiguredManager.M_Publish(AlarmList := _AlarmList);
AssertTrue(
	Condition := _AlarmList[1].MainErrorId = 0,
	Message := 'Acknowledged configured alarm must be removed in the false sample scan.'
);

TEST_FINISHED();
END_METHOD

METHOD HookOccurrencesUseTheExistingAcknowledgementLifecycle
VAR
	Alarm : ST_ExtAlarm;
	Request : ST_AlarmAckRequest;
	Accepted : BOOL;
END_VAR
VAR_INST
	bFinished : BOOL;
END_VAR
TEST('HookOccurrencesUseTheExistingAcknowledgementLifecycle');
IF bFinished THEN
	RETURN;
END_IF

Alarm.MainErrorId := 400;
Alarm.Message := 'First Hook occurrence';
Alarm.Path := 'Test.Axis';
Alarm.Severity := E_Severity.Alarm;
Alarm.DateTime := '20260912100000000';
_HookLifecycleManager.M_BeginCycle(ModuleId := 91, ConfigurationRevision := 1);
_HookLifecycleManager.M_ObserveHookAlarm(Alarm := Alarm);
_HookLifecycleManager.M_EndCycle();
_HookLifecycleManager.M_Publish(AlarmList := _AlarmList);
AssertTrue(
	Condition :=
		_AlarmList[1].ModuleId = 91
		AND _AlarmList[1].ServiceId = 0
		AND _AlarmList[1].OccurrenceCount = 1,
	Message := 'Hook lifecycle uses the Module identity and starts at one.'
);
Alarm.Message := 'Must not refresh the lifecycle snapshot';
Alarm.DateTime := '20260912100100000';
_HookLifecycleManager.M_BeginCycle(ModuleId := 91, ConfigurationRevision := 1);
_HookLifecycleManager.M_ObserveHookAlarm(Alarm := Alarm);
Accepted := _HookLifecycleManager.M_ObserveHookAlarm(Alarm := Alarm);
_HookLifecycleManager.M_EndCycle();
_HookLifecycleManager.M_Publish(AlarmList := _AlarmList);
AssertTrue(
	Condition := NOT Accepted AND _HookLifecycleManager.DuplicateId = 400,
	Message := 'Repeated submission in one scan is rejected.'
);
AssertTrue(
	Condition :=
		_AlarmList[1].OccurrenceCount = 1
		AND _AlarmList[1].Message = 'First Hook occurrence'
		AND _AlarmList[1].DateTime = '20260912100000000',
	Message := 'Continuous observation and duplicates preserve the first snapshot.'
);
_HookLifecycleManager.M_BeginCycle(ModuleId := 91, ConfigurationRevision := 1);
_HookLifecycleManager.M_EndCycle();
_HookLifecycleManager.M_Publish(AlarmList := _AlarmList);
AssertTrue(
	Condition := _AlarmList[1].MainErrorId = 400
		AND NOT _AlarmList[1].Active
		AND NOT _AlarmList[1].Acknowledged,
	Message := 'An unobserved Hook condition is inactive and latched.'
);
_HookLifecycleManager.M_BeginCycle(ModuleId := 91, ConfigurationRevision := 1);
_HookLifecycleManager.M_ObserveHookAlarm(Alarm := Alarm);
_HookLifecycleManager.M_EndCycle();
_HookLifecycleManager.M_Publish(AlarmList := _AlarmList);
AssertTrue(
	Condition := _AlarmList[1].Active
		AND NOT _AlarmList[1].Acknowledged
		AND _AlarmList[1].OccurrenceCount = 2,
	Message := 'Recurrence increments the count and clears acknowledgement.'
);

Request.Command := E_AlarmAckCommand.AcknowledgeOne;
Request.MainErrorId := 400;
Request.ServiceId := 0;
Request.RequestId := 1;
Request.bChangeRequest := TRUE;
_HookLifecycleManager.M_BeginCycle(ModuleId := 91, ConfigurationRevision := 1);
_HookLifecycleManager.M_ProcessAcknowledgement(Request := Request);
_HookLifecycleManager.M_ObserveHookAlarm(Alarm := Alarm);
_HookLifecycleManager.M_EndCycle();
_HookLifecycleManager.M_Publish(AlarmList := _AlarmList);
AssertTrue(
	Condition := _HookLifecycleManager.AckAccepted
		AND _AlarmList[1].Active
		AND _AlarmList[1].Acknowledged,
	Message := 'Acknowledging an active Hook does not remove it.'
);
Request.bChangeRequest := FALSE;
_HookLifecycleManager.M_BeginCycle(ModuleId := 91, ConfigurationRevision := 1);
_HookLifecycleManager.M_ProcessAcknowledgement(Request := Request);
_HookLifecycleManager.M_EndCycle();
_HookLifecycleManager.M_Publish(AlarmList := _AlarmList);
AssertTrue(
	Condition := _HookLifecycleManager.HookLatchedCount = 0
		AND _AlarmList[1].MainErrorId = 0,
	Message := 'The first inactive scan removes an acknowledged Hook.'
);
_HookLifecycleManager.M_BeginCycle(ModuleId := 91, ConfigurationRevision := 1);
_HookLifecycleManager.M_ObserveHookAlarm(Alarm := Alarm);
_HookLifecycleManager.M_EndCycle();
_HookLifecycleManager.M_Publish(AlarmList := _AlarmList);
AssertTrue(
	Condition :=
		_AlarmList[1].OccurrenceCount = 1
		AND NOT _AlarmList[1].Acknowledged
		AND _AlarmList[1].DateTime = '20260912100100000',
	Message := 'An occurrence after removal starts a new lifecycle.'
);

bFinished := TRUE;
TEST_FINISHED();
END_METHOD

METHOD HookAcknowledgementsRespectIdentityAndNewEventOrdering
VAR
	HookAlarm : ST_ExtAlarm;
	ServiceAlarm : ST_ExtAlarm;
	ConfiguredAlarm : ST_ExtAlarm;
	Request : ST_AlarmAckRequest;
END_VAR
VAR_INST
	bFinished : BOOL;
END_VAR
TEST('HookAcknowledgementsRespectIdentityAndNewEventOrdering');
IF bFinished THEN
	RETURN;
END_IF

HookAlarm.MainErrorId := 500;
HookAlarm.DateTime := '20260912110000000';
ServiceAlarm := HookAlarm;
ServiceAlarm.ServiceId := 11;
ConfiguredAlarm.MainErrorId := 600;
_HookAckManager.M_BeginCycle(ModuleId := 92, ConfigurationRevision := 1);
_HookAckManager.M_ObserveHookAlarm(Alarm := HookAlarm);
_HookAckManager.M_ObserveServiceAlarm(Alarm := ServiceAlarm);
_HookAckManager.M_UpdateConfiguredAlarm(
	AlarmIndex := 1,
	SampleValid := TRUE,
	ConditionMet := TRUE,
	Alarm := ConfiguredAlarm,
	UtcDateTime := '20260912110000000'
);
_HookAckManager.M_EndCycle();
_HookAckManager.M_Publish(AlarmList := _AlarmList);
AssertTrue(
	Condition :=
		_AlarmList[1].ServiceId = 11
		AND _AlarmList[2].MainErrorId = 600
		AND _AlarmList[3].MainErrorId = 500,
	Message := 'Publish order is Service, JSON, Hook; matching numbers may coexist.'
);
Request.Command := E_AlarmAckCommand.AcknowledgeOne;
Request.ServiceId := 0;
Request.MainErrorId := 500;
Request.RequestId := 1;
Request.bChangeRequest := TRUE;
_HookAckManager.M_BeginCycle(ModuleId := 92, ConfigurationRevision := 1);
_HookAckManager.M_ProcessAcknowledgement(Request := Request);
_HookAckManager.M_ObserveHookAlarm(Alarm := HookAlarm);
_HookAckManager.M_ObserveServiceAlarm(Alarm := ServiceAlarm);
_HookAckManager.M_EndCycle();
_HookAckManager.M_Publish(AlarmList := _AlarmList);
AssertTrue(
	Condition :=
		_HookAckManager.AckAccepted
		AND _AlarmList[3].Acknowledged
		AND NOT _AlarmList[1].Acknowledged
		AND NOT _AlarmList[2].Acknowledged,
	Message := 'AcknowledgeOne targets the composite identity, not just the error number.'
);
Request.bChangeRequest := FALSE;
_HookAckManager.M_BeginCycle(ModuleId := 92, ConfigurationRevision := 1);
_HookAckManager.M_ProcessAcknowledgement(Request := Request);
_HookAckManager.M_ObserveHookAlarm(Alarm := HookAlarm);
_HookAckManager.M_ObserveServiceAlarm(Alarm := ServiceAlarm);
_HookAckManager.M_EndCycle();
_HookAckManager.M_Publish(AlarmList := _AlarmList);
Request.Command := E_AlarmAckCommand.AcknowledgeAll;
Request.RequestId := 2;
Request.bChangeRequest := TRUE;
_HookAckManager.M_BeginCycle(ModuleId := 92, ConfigurationRevision := 1);
_HookAckManager.M_ProcessAcknowledgement(Request := Request);
_HookAckManager.M_ObserveHookAlarm(Alarm := HookAlarm);
_HookAckManager.M_ObserveServiceAlarm(Alarm := ServiceAlarm);
HookAlarm.MainErrorId := 501;
_HookAckManager.M_ObserveHookAlarm(Alarm := HookAlarm);
_HookAckManager.M_EndCycle();
_HookAckManager.M_Publish(AlarmList := _AlarmList);
AssertTrue(
	Condition := _AlarmList[1].Acknowledged
		AND _AlarmList[2].Acknowledged
		AND _AlarmList[3].Acknowledged,
	Message := 'AcknowledgeAll includes all three existing sources.'
);
AssertTrue(
	Condition := _AlarmList[4].MainErrorId = 501 AND NOT _AlarmList[4].Acknowledged,
	Message := 'AcknowledgeAll cannot consume a new Hook event in the same scan.'
);
Request.bChangeRequest := FALSE;
_HookAckManager.M_BeginCycle(ModuleId := 92, ConfigurationRevision := 1);
_HookAckManager.M_ProcessAcknowledgement(Request := Request);
_HookAckManager.M_UpdateConfiguredAlarm(
	AlarmIndex := 1,
	SampleValid := TRUE,
	ConditionMet := FALSE,
	Alarm := ConfiguredAlarm,
	UtcDateTime := '20260912110100000'
);
_HookAckManager.M_EndCycle();
_HookAckManager.M_Publish(AlarmList := _AlarmList);
AssertTrue(
	Condition :=
		_HookAckManager.ServiceLatchedCount = 0
		AND _HookAckManager.ConfiguredLatchedCount = 0
		AND _HookAckManager.HookLatchedCount = 1,
	Message := 'Inactive acknowledged identities are removed from all sources.'
);
AssertTrue(
	Condition := _AlarmList[1].MainErrorId = 501 AND NOT _AlarmList[1].Active,
	Message := 'The new unacknowledged Hook event remains latched.'
);

// Acknowledge an inactive identity before its next observation: start a fresh lifecycle.
Request.Command := E_AlarmAckCommand.AcknowledgeOne;
Request.MainErrorId := 501;
Request.RequestId := 3;
Request.bChangeRequest := TRUE;
_HookAckManager.M_BeginCycle(ModuleId := 92, ConfigurationRevision := 1);
_HookAckManager.M_ProcessAcknowledgement(Request := Request);
_HookAckManager.M_ObserveHookAlarm(Alarm := HookAlarm);
_HookAckManager.M_EndCycle();
_HookAckManager.M_Publish(AlarmList := _AlarmList);
AssertTrue(
	Condition :=
		_AlarmList[1].MainErrorId = 501
		AND _AlarmList[1].Active
		AND NOT _AlarmList[1].Acknowledged
		AND _AlarmList[1].OccurrenceCount = 1,
	Message :=
		'Acknowledgement before a new observation cannot pre-acknowledge the new lifecycle.'
);

bFinished := TRUE;
TEST_FINISHED();
END_METHOD

METHOD HookCapacityAndConfigurationOwnershipHaveSeparateResetScopes
VAR
	Alarm : ST_ExtAlarm;
	Request : ST_AlarmAckRequest;
	nIndex : UINT;
	Accepted : BOOL;
END_VAR
VAR_INST
	bFinished : BOOL;
END_VAR
TEST('HookCapacityAndConfigurationOwnershipHaveSeparateResetScopes');
IF bFinished THEN
	RETURN;
END_IF

AssertTrue(
	Condition :=
		Param_Config.MaxConfiguredAlarmsPerModule = 30
		AND Param_Config.MaxHookAlarmsPerModule = 30
		AND Param_Config.MaxServiceAlarmsPerModule = 40
		AND Param_Config.MaxPublishedModuleAlarms = 100,
	Message := 'Alarm partitions are fixed at JSON 30, Hook 30, Service 40.'
);
_HookCapacityManager.M_BeginCycle(ModuleId := 93, ConfigurationRevision := 1);
FOR nIndex := 1 TO Param_Config.MaxConfiguredAlarmsPerModule DO
	Alarm.MainErrorId := 1000 + UINT_TO_UDINT(nIndex);
	_HookCapacityManager.M_UpdateConfiguredAlarm(
		AlarmIndex := nIndex,
		SampleValid := TRUE,
		ConditionMet := TRUE,
		Alarm := Alarm,
		UtcDateTime := '20260912120000000'
	);
END_FOR
Alarm.ServiceId := 0;
FOR nIndex := 1 TO Param_Config.MaxHookAlarmsPerModule DO
	Alarm.MainErrorId := 2000 + UINT_TO_UDINT(nIndex);
	_HookCapacityManager.M_ObserveHookAlarm(Alarm := Alarm);
END_FOR
Alarm.ServiceId := 11;
FOR nIndex := 1 TO Param_Config.MaxServiceAlarmsPerModule DO
	Alarm.MainErrorId := 3000 + UINT_TO_UDINT(nIndex);
	_HookCapacityManager.M_ObserveServiceAlarm(Alarm := Alarm);
END_FOR
_HookCapacityManager.M_EndCycle();
_HookCapacityManager.M_Publish(AlarmList := _AlarmList);
AssertTrue(
	Condition :=
		_HookCapacityManager.ConfiguredLatchedCount = 30
		AND _HookCapacityManager.HookLatchedCount = 30
		AND _HookCapacityManager.ServiceLatchedCount = 40
		AND NOT _HookCapacityManager.Overflow,
	Message := 'All reserved capacities can be filled simultaneously.'
);
AssertTrue(
	Condition :=
		_AlarmList[40].MainErrorId = 3040
		AND _AlarmList[70].MainErrorId = 1030
		AND _AlarmList[100].MainErrorId = 2030,
	Message := 'All 100 entries preserve the source ordering.'
);
Alarm.MainErrorId := 9999;
Accepted := _HookCapacityManager.M_ObserveServiceAlarm(Alarm := Alarm);
AssertTrue(
	Condition := NOT Accepted,
	Message := 'The 41st Service lifecycle is rejected.'
);
Alarm.ServiceId := 0;
Accepted := _HookCapacityManager.M_ObserveHookAlarm(Alarm := Alarm);
AssertTrue(Condition := NOT Accepted, Message := 'The 31st Hook lifecycle is rejected.');
_HookCapacityManager.M_Publish(AlarmList := _AlarmList);
AssertTrue(
	Condition := _HookCapacityManager.Overflow AND _AlarmList[100].MainErrorId = 2030,
	Message := 'Overflow cannot overwrite a latched Hook identity.'
);
_HookCapacityManager.M_BeginCycle(ModuleId := 93, ConfigurationRevision := 2);
_HookCapacityManager.M_SuppressHookAlarm(MainErrorId := 2001);
_HookCapacityManager.M_EndCycle();
_HookCapacityManager.M_Publish(AlarmList := _AlarmList);
AssertTrue(
	Condition :=
		_HookCapacityManager.ConfiguredLatchedCount = 0
		AND _HookCapacityManager.HookLatchedCount = 29
		AND _HookCapacityManager.ServiceLatchedCount = 40
		AND NOT _HookCapacityManager.Overflow,
	Message :=
		'Revision resets JSON and only the explicitly overridden Hook; Services survive.'
);
AssertTrue(
	Condition := _AlarmList[41].MainErrorId = 2002 AND NOT _AlarmList[41].Active,
	Message := 'Unrelated unacknowledged Hook lifecycles survive revisions.'
);
// Suppressed Hook lifecycles cannot be acknowledged through a stale identity.
Request.Command := E_AlarmAckCommand.AcknowledgeOne;
Request.MainErrorId := 2001;
Request.RequestId := 1;
Request.bChangeRequest := TRUE;
_HookCapacityManager.M_ProcessAcknowledgement(Request := Request);
AssertTrue(
	Condition :=
		NOT _HookCapacityManager.AckAccepted
		AND _HookCapacityManager.AckError = E_AlarmAckError.AlarmNotFound,
	Message := 'A JSON takeover removes the old Hook identity before acknowledgement.'
);
_HookCapacityManager.M_BeginCycle(ModuleId := 94, ConfigurationRevision := 2);
_HookCapacityManager.M_EndCycle();
_HookCapacityManager.M_Publish(AlarmList := _AlarmList);
AssertTrue(
	Condition :=
		_HookCapacityManager.ConfiguredLatchedCount = 0
		AND _HookCapacityManager.HookLatchedCount = 0
		AND _HookCapacityManager.ServiceLatchedCount = 0
		AND _HookCapacityManager.AckResponseId = 0,
	Message := 'Changing Module identity clears every lifecycle and acknowledgement.'
);

bFinished := TRUE;
TEST_FINISHED();
END_METHOD

END_FUNCTION_BLOCK

// ---- POUs/Test Suites/Module/FB_ModuleBaseTests.TcPOU
FUNCTION_BLOCK FB_ModuleBaseTests EXTENDS TcUnit.FB_TestSuite
VAR
	// Keep the large Module instance at Test Suite scope to avoid Method stack overflow.
	HeartbeatModule : FB_TestableModuleBase;
	HookModule : FB_TestableHookModule;
	OverrideModule : FB_TestableHookModule;
	CapacityModule : FB_TestableHookModule;
	RegressionModule : FB_TestableModuleBase;
END_VAR

EmptyHooksPreserveConfiguredDataAndServiceAggregation();
HookAndVariableCapacitiesPreserveExistingEntries();
JsonOwnsHookIdentitiesIncludingFalseAndInvalidSamples();
HooksReadBaseUnitAfterUpdateAndEnforceSubmissionContract();
HeartbeatChangeResetsTimeoutAndRestoresControlSource();

METHOD HeartbeatChangeResetsTimeoutAndRestoresControlSource
VAR_INST
	ModuleCtrl : ST_ModuleCtrl;
	SystemContext : ST_SystemContext;
	RuntimeConfig : ST_ModuleRuntimeConfig;
	VariableNodeReader : FB_LinkVariableManager;
	HeartbeatIndex : UDINT;
	PhaseTimer : TON;
	WatchdogTimer : TON;
	nPhase : UINT;
END_VAR
TEST('HeartbeatChangeResetsTimeoutAndRestoresControlSource');

CASE nPhase OF
	0:
		SystemContext.ModuleHeartbeatTimeout := T#50MS;
		HeartbeatIndex := 100;
		HeartbeatModule(
			ModuleCtrl := ModuleCtrl,
			SystemContext := SystemContext,
			HeartbeatIndex := HeartbeatIndex,
			RuntimeConfig := RuntimeConfig,
			VariableNodeReader := VariableNodeReader);
		AssertTrue(
			Condition := HeartbeatModule.ModuleStatus.IsControlSourceAlive,
			Message := 'A changed HeartbeatIndex must publish an alive Control Source.');
		PhaseTimer(IN := FALSE, PT := T#30MS);
		WatchdogTimer(IN := FALSE, PT := T#100MS);
		nPhase := 1;

	1:
		// Hold the first index for less than the injected timeout.
		HeartbeatModule(
			ModuleCtrl := ModuleCtrl,
			SystemContext := SystemContext,
			HeartbeatIndex := HeartbeatIndex,
			RuntimeConfig := RuntimeConfig,
			VariableNodeReader := VariableNodeReader);
		PhaseTimer(IN := TRUE, PT := T#30MS);
		AssertTrue(
			Condition := HeartbeatModule.ModuleStatus.IsControlSourceAlive,
			Message := 'An unchanged HeartbeatIndex must remain alive before its timeout.');
		IF PhaseTimer.Q THEN
			PhaseTimer(IN := FALSE, PT := T#30MS);
			HeartbeatIndex := 101;
			nPhase := 2;
		END_IF

	2:
		// A new index must reset the heartbeat timeout in the same Module scan.
		HeartbeatModule(
			ModuleCtrl := ModuleCtrl,
			SystemContext := SystemContext,
			HeartbeatIndex := HeartbeatIndex,
			RuntimeConfig := RuntimeConfig,
			VariableNodeReader := VariableNodeReader);
		AssertTrue(
			Condition := HeartbeatModule.ModuleStatus.IsControlSourceAlive,
			Message := 'A new HeartbeatIndex must reset the timeout immediately.');
		PhaseTimer(IN := FALSE, PT := T#30MS);
		nPhase := 3;

	3:
		// The total time since the first index stopped changing now exceeds 50 ms,
		// while the latest index has remained unchanged for only 30 ms.
		HeartbeatModule(
			ModuleCtrl := ModuleCtrl,
			SystemContext := SystemContext,
			HeartbeatIndex := HeartbeatIndex,
			RuntimeConfig := RuntimeConfig,
			VariableNodeReader := VariableNodeReader);
		PhaseTimer(IN := TRUE, PT := T#30MS);
		AssertTrue(
			Condition := HeartbeatModule.ModuleStatus.IsControlSourceAlive,
			Message := 'The reset timeout must remain alive for its own pre-timeout interval.');
		IF PhaseTimer.Q THEN
			PhaseTimer(IN := FALSE, PT := T#30MS);
			WatchdogTimer(IN := FALSE, PT := T#100MS);
			nPhase := 4;
		END_IF

	4:
		// Keep the second index stable until the injected timeout expires.
		HeartbeatModule(
			ModuleCtrl := ModuleCtrl,
			SystemContext := SystemContext,
			HeartbeatIndex := HeartbeatIndex,
			RuntimeConfig := RuntimeConfig,
			VariableNodeReader := VariableNodeReader);
		WatchdogTimer(IN := TRUE, PT := T#100MS);
		IF HeartbeatModule.ModuleStatus.IsControlSourceAlive THEN
			IF WatchdogTimer.Q THEN
				AssertTrue(
					Condition := FALSE,
					Message := 'A stable HeartbeatIndex must time out before the watchdog expires.');
				PhaseTimer(IN := FALSE, PT := T#30MS);
				WatchdogTimer(IN := FALSE, PT := T#100MS);
				SystemContext.ModuleHeartbeatTimeout := T#0S;
				HeartbeatIndex := 0;
				nPhase := 0;
				TEST_FINISHED();
			END_IF
		ELSE
			AssertFalse(
				Condition := HeartbeatModule.ModuleStatus.IsControlSourceAlive,
				Message :=
					'A stable HeartbeatIndex must publish a dead Control Source after timeout.');
			WatchdogTimer(IN := FALSE, PT := T#100MS);
			nPhase := 5;
		END_IF

	5:
		// The next changed index must recover the public status immediately.
		HeartbeatIndex := 102;
		HeartbeatModule(
			ModuleCtrl := ModuleCtrl,
			SystemContext := SystemContext,
			HeartbeatIndex := HeartbeatIndex,
			RuntimeConfig := RuntimeConfig,
			VariableNodeReader := VariableNodeReader);
		AssertTrue(
			Condition := HeartbeatModule.ModuleStatus.IsControlSourceAlive,
			Message :=
				'A changed HeartbeatIndex must recover a timed-out Control Source immediately.');

		PhaseTimer(IN := FALSE, PT := T#30MS);
		WatchdogTimer(IN := FALSE, PT := T#100MS);
		SystemContext.ModuleHeartbeatTimeout := T#0S;
		HeartbeatIndex := 0;
		nPhase := 0;
		TEST_FINISHED();
END_CASE
END_METHOD

METHOD HooksReadBaseUnitAfterUpdateAndEnforceSubmissionContract
VAR_INST
	Ctrl : ST_ModuleCtrl;
	Context : ST_SystemContext;
	Config : ST_ModuleRuntimeConfig;
	Axis : FB_FakeAxis_BaseUnit;
	Reader : FB_FakeHookValueReader;
END_VAR
VAR_INST
	bFinished : BOOL;
END_VAR
TEST('HooksReadBaseUnitAfterUpdateAndEnforceSubmissionContract');
IF bFinished THEN
	RETURN;
END_IF

Config.ModuleId := 81;
Config.Valid := TRUE;
Config.Enabled := TRUE;
Config.Revision := 1;
Context.UtcDateTime := '20260912090000000';
Axis.M_SetAxisState(Disabled := TRUE, HasJob := FALSE);
Axis.M_SetAxisFeedback(ActualPosition := 12.5, ActualVelocity := 0);
HookModule.ProbeInvalidCalls := TRUE;
HookModule.DuplicateAlarm := TRUE;
HookModule.DuplicateVariable := TRUE;
HookModule(
	ModuleCtrl := Ctrl,
	SystemContext := Context,
	RuntimeConfig := Config,
	VariableNodeReader := Reader,
	Axis := Axis
);
AssertTrue(
	Condition :=
		HookModule.BaseUnitScans = 1
		AND HookModule.AlarmHookScans = 1
		AND HookModule.VariableHookScans = 1,
	Message := 'Both hooks run once outside Execute.'
);
AssertTrue(
	Condition :=
		HookModule.AlarmObservedScan = HookModule.BaseUnitScans
		AND HookModule.VariableObservedScan = HookModule.BaseUnitScans,
	Message := 'Hooks follow the Base Unit update.'
);
AssertTrue(
	Condition := Axis.CurrentCycle = 1,
	Message := 'The typed Base Unit has completed its cyclic update.'
);
AssertTrue(
	Condition := HookModule.AlarmAccepted AND HookModule.VariableAccepted,
	Message := 'Valid Hook submissions are accepted.'
);
AssertTrue(
	Condition :=
		NOT HookModule.OutsideAlarmAccepted
		AND NOT HookModule.OutsideVariableAccepted
		AND NOT HookModule.CrossAlarmAccepted
		AND NOT HookModule.CrossVariableAccepted,
	Message := 'Wrong submission phases are rejected.'
);
AssertTrue(
	Condition := NOT HookModule.ZeroAlarmAccepted AND NOT HookModule.ZeroVariableAccepted,
	Message := 'Zero identities are rejected within the right hook.'
);
AssertTrue(
	Condition := NOT HookModule.DuplicateAlarmAccepted
		AND NOT HookModule.DuplicateVariableAccepted,
	Message := 'Second Hook submissions are rejected.'
);
AssertTrue(
	Condition :=
		HookModule.ModuleStatus.Alarm.DuplicateId = 9001
		AND HookModule.ModuleStatus.Variable.DuplicateId = 8001,
	Message := 'First duplicate identities are published.'
);
AssertTrue(
	Condition :=
		HookModule.ModuleAlarmList[1].Message = 'Axis disabled'
		AND HookModule.ModuleVariableList[1].Name = 'Axis position',
	Message := 'Duplicate submissions preserve the first descriptors.'
);
AssertTrue(
	Condition := HookModule.ModuleAlarmList[1].ModuleId = 81
		AND HookModule.ModuleAlarmList[1].ServiceId = 0,
	Message := 'The framework stamps the Module identity.'
);
AssertTrue(
	Condition :=
		HookModule.ModuleAlarmList[1].DateTime = Context.UtcDateTime
		AND HookModule.ModuleAlarmList[1].OccurrenceCount = 1,
	Message := 'The framework stamps the first occurrence.'
);
AssertTrue(
	Condition := HookModule.ModuleVariableList[1].Value = LREAL_TO_STRING(12.5),
	Message := 'The SVID reads Axis feedback directly.'
);
HookModule.DuplicateAlarm := FALSE;
HookModule.DuplicateVariable := FALSE;
Axis.M_SetAxisFeedback(ActualPosition := 25.0, ActualVelocity := 0);
HookModule(
	ModuleCtrl := Ctrl,
	SystemContext := Context,
	RuntimeConfig := Config,
	VariableNodeReader := Reader,
	Axis := Axis
);
AssertTrue(
	Condition := HookModule.ModuleVariableList[1].Value = LREAL_TO_STRING(25.0),
	Message := 'The Hook SVID changes in the next Module scan.'
);
AssertTrue(
	Condition := HookModule.ModuleAlarmList[1].OccurrenceCount = 1,
	Message := 'Continuous active scans do not count as recurrences.'
);
AssertTrue(
	Condition :=
		HookModule.ModuleStatus.Alarm.DuplicateId = 0
		AND HookModule.ModuleStatus.Variable.DuplicateId = 0,
	Message := 'Duplicate diagnostics reset each scan.'
);
HookModule.VariableCount := 0;
Axis.M_SetAxisState(Disabled := FALSE, HasJob := FALSE);
HookModule(
	ModuleCtrl := Ctrl,
	SystemContext := Context,
	RuntimeConfig := Config,
	VariableNodeReader := Reader,
	Axis := Axis
);
AssertTrue(
	Condition := HookModule.ModuleStatus.Variable.PublishedCount = 0
		AND HookModule.ModuleVariableList[1].Id = 0,
	Message := 'Omitted SVIDs disappear without stale values.'
);
AssertTrue(
	Condition := HookModule.ModuleStatus.Alarm.HookLatchedCount = 1
		AND NOT HookModule.ModuleAlarmList[1].Active,
	Message := 'Omitted alarms become inactive but remain latched.'
);
Ctrl.AlarmAckRequest.Command := E_AlarmAckCommand.AcknowledgeOne;
Ctrl.AlarmAckRequest.MainErrorId := 9001;
Ctrl.AlarmAckRequest.ServiceId := 0;
Ctrl.AlarmAckRequest.RequestId := 1;
Ctrl.AlarmAckRequest.bChangeRequest := TRUE;
HookModule(
	ModuleCtrl := Ctrl,
	SystemContext := Context,
	RuntimeConfig := Config,
	VariableNodeReader := Reader,
	Axis := Axis
);
AssertTrue(
	Condition :=
		HookModule.ModuleStatus.Alarm.AckAccepted
		AND HookModule.ModuleStatus.Alarm.HookLatchedCount = 0,
	Message := 'Module acknowledgement removes an inactive Hook lifecycle.'
);

bFinished := TRUE;
TEST_FINISHED();
END_METHOD

METHOD JsonOwnsHookIdentitiesIncludingFalseAndInvalidSamples
VAR_INST
	Ctrl : ST_ModuleCtrl;
	Context : ST_SystemContext;
	Config : ST_ModuleRuntimeConfig;
	Axis : FB_FakeAxis_BaseUnit;
	Reader : FB_FakeHookValueReader;
END_VAR
VAR_INST
	bFinished : BOOL;
END_VAR
TEST('JsonOwnsHookIdentitiesIncludingFalseAndInvalidSamples');
IF bFinished THEN
	RETURN;
END_IF

Config.ModuleId := 82;
Config.Enabled := TRUE;
Config.Valid := TRUE;
Config.Revision := 1;
OverrideModule.AlarmCount := 2;
Axis.M_SetAxisState(Disabled := TRUE, HasJob := FALSE);
Axis.M_SetAxisFeedback(ActualPosition := 12.5, ActualVelocity := 0);
OverrideModule(
	ModuleCtrl := Ctrl,
	SystemContext := Context,
	RuntimeConfig := Config,
	VariableNodeReader := Reader,
	Axis := Axis
);
AssertTrue(
	Condition := OverrideModule.ModuleStatus.Alarm.HookLatchedCount = 2,
	Message := 'Two Hook identities are initially active.'
);

// A new JSON definition takes ownership even while its condition is false.
Config.Revision := 2;
Config.AlarmCount := 1;
Config.AlarmBindings[1].NodeHandle := 1;
Config.AlarmBindings[1].Definition.MainErrorId := 9001;
Config.AlarmBindings[1].Definition.SourceErrorId := 77;
Config.AlarmBindings[1].Definition.Source := 'Test.JsonSource';
Config.AlarmBindings[1].Definition.DataType := E_ConfigDataType.Float64;
Config.AlarmBindings[1].Definition.Operator := E_AlarmOperator.GreaterThan;
Config.AlarmBindings[1].Definition.Threshold := 10.0;
Config.AlarmBindings[1].Definition.Message := 'JSON owns this alarm';
Config.AlarmBindings[1].Definition.Severity := E_Severity.Warning;
Config.VariableCount := 1;
Config.VariableBindings[1].NodeHandle := 1;
Config.VariableBindings[1].Definition.Id := 8001;
Config.VariableBindings[1].Definition.Name := 'JSON value';
Config.VariableBindings[1].Definition.Unit := 'rpm';
Config.VariableBindings[1].Definition.DataType := E_ConfigDataType.Integer32;
Reader.Sample := 5.0;
OverrideModule.DuplicateAlarm := TRUE;
OverrideModule.DuplicateVariable := TRUE;
OverrideModule(
	ModuleCtrl := Ctrl,
	SystemContext := Context,
	RuntimeConfig := Config,
	VariableNodeReader := Reader,
	Axis := Axis
);
AssertTrue(
	Condition :=
		OverrideModule.ModuleStatus.Alarm.ConfiguredLatchedCount = 0
		AND OverrideModule.ModuleStatus.Alarm.HookLatchedCount = 1,
	Message := 'JSON false suppresses the matching Hook and preserves other lifecycles.'
);
AssertTrue(
	Condition :=
		OverrideModule.ModuleAlarmList[1].MainErrorId = 9002
		AND OverrideModule.ModuleAlarmList[1].OccurrenceCount = 1,
	Message := 'Revision changes preserve unrelated Hook occurrences.'
);
AssertTrue(
	Condition := OverrideModule.DuplicateAlarmAccepted
		AND OverrideModule.DuplicateVariableAccepted,
	Message := 'JSON ownership is accepted without consuming Hook capacity.'
);
AssertTrue(
	Condition :=
		OverrideModule.ModuleStatus.Alarm.DuplicateId = 0
		AND OverrideModule.ModuleStatus.Variable.DuplicateId = 0,
	Message := 'Repeated JSON-owned submissions are not duplicate errors.'
);
AssertTrue(
	Condition :=
		OverrideModule.ModuleVariableList[1].Name = 'JSON value'
		AND OverrideModule.ModuleVariableList[1].Unit = 'rpm'
		AND OverrideModule.ModuleVariableList[1].Value = '5'
		AND OverrideModule.ModuleVariableList[1].DataType = E_DescriptorType.Integer_32bit,
	Message := 'JSON owns the complete SVID descriptor and value.'
);

// Invalid samples never fall back to a true Hook condition or its SVID value.
Reader.SampleValid := FALSE;
OverrideModule(
	ModuleCtrl := Ctrl,
	SystemContext := Context,
	RuntimeConfig := Config,
	VariableNodeReader := Reader,
	Axis := Axis
);
AssertTrue(
	Condition :=
		OverrideModule.ModuleStatus.Alarm.ConfiguredLatchedCount = 0
		AND OverrideModule.ModuleStatus.Alarm.HookLatchedCount = 1,
	Message := 'Invalid JSON samples do not resurrect the overridden Hook.'
);
AssertTrue(
	Condition :=
		OverrideModule.ModuleVariableList[1].Value = ''
		AND OverrideModule.ModuleVariableList[1].Name = 'JSON value',
	Message :=
		'Invalid JSON SVID reads keep JSON metadata and the existing empty-value behavior.'
);
Reader.SampleValid := TRUE;
Reader.Sample := 20.0;
OverrideModule(
	ModuleCtrl := Ctrl,
	SystemContext := Context,
	RuntimeConfig := Config,
	VariableNodeReader := Reader,
	Axis := Axis
);
AssertTrue(
	Condition :=
		OverrideModule.ModuleStatus.Alarm.ConfiguredLatchedCount = 1
		AND OverrideModule.ModuleStatus.Alarm.HookLatchedCount = 1,
	Message := 'The JSON condition alone starts its lifecycle.'
);
AssertTrue(
	Condition :=
		OverrideModule.ModuleAlarmList[1].MainErrorId = 9001
		AND OverrideModule.ModuleAlarmList[1].Message = 'JSON owns this alarm'
		AND OverrideModule.ModuleAlarmList[1].Severity = E_Severity.Warning
		AND OverrideModule.ModuleAlarmList[1].SourceErrorId = 77,
	Message :=
		'JSON replaces the complete Alarm definition before the remaining Hook is published.'
);
Reader.SampleValid := FALSE;
OverrideModule(
	ModuleCtrl := Ctrl,
	SystemContext := Context,
	RuntimeConfig := Config,
	VariableNodeReader := Reader,
	Axis := Axis
);
AssertTrue(
	Condition :=
		OverrideModule.ModuleAlarmList[1].Active
		AND OverrideModule.ModuleAlarmList[1].OccurrenceCount = 1,
	Message := 'Invalid JSON samples retain the last lifecycle state.'
);

// A removed override lets the Hook start a fresh lifecycle.
Config.Revision := 3;
Config.AlarmCount := 0;
Config.VariableCount := 0;
Reader.SampleValid := TRUE;
OverrideModule.DuplicateAlarm := FALSE;
OverrideModule.DuplicateVariable := FALSE;
OverrideModule(
	ModuleCtrl := Ctrl,
	SystemContext := Context,
	RuntimeConfig := Config,
	VariableNodeReader := Reader,
	Axis := Axis
);
AssertTrue(
	Condition :=
		OverrideModule.ModuleStatus.Alarm.ConfiguredLatchedCount = 0
		AND OverrideModule.ModuleStatus.Alarm.HookLatchedCount = 2,
	Message := 'Removing JSON ownership re-enables Hook submission.'
);
AssertTrue(
	Condition := OverrideModule.ModuleVariableList[1].Name = 'Axis position',
	Message := 'Removing JSON ownership re-enables the Hook SVID.'
);
Config.Valid := FALSE;
OverrideModule.VariableCount := 0;
OverrideModule(
	ModuleCtrl := Ctrl,
	SystemContext := Context,
	RuntimeConfig := Config,
	VariableNodeReader := Reader,
	Axis := Axis
);
AssertTrue(
	Condition :=
		OverrideModule.ModuleStatus.Variable.PublishedCount = 0
		AND OverrideModule.ModuleVariableList[1].Id = 0,
	Message := 'Invalid configuration cannot retain stale SVID entries.'
);

bFinished := TRUE;
TEST_FINISHED();
END_METHOD

METHOD HookAndVariableCapacitiesPreserveExistingEntries
VAR_INST
	Ctrl : ST_ModuleCtrl;
	Context : ST_SystemContext;
	Config : ST_ModuleRuntimeConfig;
	Axis : FB_FakeAxis_BaseUnit;
	Reader : FB_FakeHookValueReader;
END_VAR
VAR
	nIndex : UINT;
END_VAR
VAR_INST
	bFinished : BOOL;
END_VAR
TEST('HookAndVariableCapacitiesPreserveExistingEntries');
IF bFinished THEN
	RETURN;
END_IF

Config.ModuleId := 83;
Config.Valid := TRUE;
Config.Enabled := TRUE;
Config.Revision := 1;
Axis.M_SetAxisState(Disabled := TRUE, HasJob := FALSE);
CapacityModule.AlarmCount := Param_Config.MaxHookAlarmsPerModule + 1;
CapacityModule.VariableCount := Param_Config.MaxModuleVariable + 1;
CapacityModule(
	ModuleCtrl := Ctrl,
	SystemContext := Context,
	RuntimeConfig := Config,
	VariableNodeReader := Reader,
	Axis := Axis
);
AssertTrue(
	Condition :=
		CapacityModule.ModuleStatus.Alarm.HookLatchedCount = 30
		AND CapacityModule.ModuleStatus.Alarm.Overflow
		AND NOT CapacityModule.AlarmAccepted,
	Message := 'The 31st Hook lifecycle is rejected without replacing an existing one.'
);
AssertTrue(
	Condition :=
		CapacityModule.ModuleStatus.Variable.PublishedCount = 100
		AND CapacityModule.ModuleStatus.Variable.Overflow
		AND NOT CapacityModule.VariableAccepted,
	Message := 'The 101st SVID is rejected without replacing an existing one.'
);
AssertTrue(
	Condition :=
		CapacityModule.ModuleAlarmList[30].MainErrorId = 9030
		AND CapacityModule.ModuleAlarmList[31].MainErrorId = 0,
	Message := 'Hook overflow preserves its last available slot.'
);
AssertTrue(
	Condition := CapacityModule.ModuleVariableList[100].Id = 8100,
	Message := 'Variable overflow preserves its last available slot.'
);
// Filling all SVID positions with JSON leaves no space for Hook-only identities.
Config.VariableCount := Param_Config.MaxModuleVariable;
FOR nIndex := 1 TO Config.VariableCount DO
	Config.VariableBindings[nIndex].Definition.Id := 10000 + UINT_TO_UDINT(nIndex);
	Config.VariableBindings[nIndex].Definition.DataType := E_ConfigDataType.Float64;
	Config.VariableBindings[nIndex].NodeHandle := 1;
END_FOR
CapacityModule.AlarmCount := 1;
CapacityModule.VariableCount := 1;
CapacityModule(
	ModuleCtrl := Ctrl,
	SystemContext := Context,
	RuntimeConfig := Config,
	VariableNodeReader := Reader,
	Axis := Axis
);
AssertTrue(
	Condition :=
		NOT CapacityModule.ModuleStatus.Alarm.Overflow
		AND CapacityModule.ModuleStatus.Variable.Overflow,
	Message := 'Overflow diagnostics reset independently each scan.'
);
AssertTrue(
	Condition := CapacityModule.ModuleVariableList[100].Id = 10100,
	Message := 'JSON takes capacity before Hook submissions.'
);
Config.VariableBindings[1].Definition.Id := 8001;
CapacityModule(
	ModuleCtrl := Ctrl,
	SystemContext := Context,
	RuntimeConfig := Config,
	VariableNodeReader := Reader,
	Axis := Axis
);
AssertTrue(
	Condition :=
		CapacityModule.VariableAccepted
		AND NOT CapacityModule.ModuleStatus.Variable.Overflow
		AND CapacityModule.ModuleStatus.Variable.PublishedCount = 100,
	Message := 'A JSON-owned Hook ID needs no extra slot even when full.'
);
Config.VariableCount := 99;
Config.VariableBindings[1].Definition.Id := 10001;
CapacityModule(
	ModuleCtrl := Ctrl,
	SystemContext := Context,
	RuntimeConfig := Config,
	VariableNodeReader := Reader,
	Axis := Axis
);
AssertTrue(
	Condition :=
		CapacityModule.ModuleStatus.Variable.PublishedCount = 100
		AND CapacityModule.ModuleVariableList[100].Id = 8001
		AND NOT CapacityModule.ModuleStatus.Variable.Overflow,
	Message := 'Hook SVIDs use the remaining combined capacity.'
);

bFinished := TRUE;
TEST_FINISHED();
END_METHOD

METHOD EmptyHooksPreserveConfiguredDataAndServiceAggregation
VAR_INST
	Ctrl : ST_ModuleCtrl;
	Context : ST_SystemContext;
	Config : ST_ModuleRuntimeConfig;
	Reader : FB_FakeHookValueReader;
	ServiceStatus : ST_ServiceStatus;
	bFinished : BOOL;
END_VAR
TEST('EmptyHooksPreserveConfiguredDataAndServiceAggregation');

IF bFinished THEN
	RETURN;
END_IF
Config.ModuleId := 84;
Config.Valid := TRUE;
Config.Enabled := TRUE;
Config.Revision := 1;
Config.VariableCount := 1;
Config.VariableBindings[1].Definition.Id := 8001;
Config.VariableBindings[1].Definition.Name := 'Configured variable';
Config.VariableBindings[1].Definition.DataType := E_ConfigDataType.Float64;
Config.VariableBindings[1].NodeHandle := 1;
Config.AlarmCount := 1;
Config.AlarmBindings[1].Definition.MainErrorId := 9001;
Config.AlarmBindings[1].Definition.Message := 'Configured alarm';
Config.AlarmBindings[1].Definition.DataType := E_ConfigDataType.Float64;
Config.AlarmBindings[1].Definition.Operator := E_AlarmOperator.GreaterThan;
Config.AlarmBindings[1].Definition.Threshold := 10.0;
Config.AlarmBindings[1].NodeHandle := 1;
Reader.Sample := 42.0;
ServiceStatus.ErrorList[1].MainErrorId := 9001;
ServiceStatus.ErrorList[1].ServiceId := 11;
ServiceStatus.ErrorList[1].Message := 'Service alarm';
ServiceStatus.Data.DataList[1].Id := 7001;
ServiceStatus.Data.DataList[1].Name := 'Completed result';
ServiceStatus.Data.DataList[1].DataType := E_DescriptorType.Integer_32bit;
ServiceStatus.Data.DataList[1].Value := '123';
RegressionModule.M_SetServiceStatus(Status := ServiceStatus);
RegressionModule(
	ModuleCtrl := Ctrl,
	SystemContext := Context,
	RuntimeConfig := Config,
	VariableNodeReader := Reader
);
AssertTrue(
	Condition :=
		RegressionModule.ModuleStatus.Alarm.HookLatchedCount = 0
		AND RegressionModule.ModuleStatus.Alarm.ConfiguredLatchedCount = 1
		AND RegressionModule.ModuleStatus.Alarm.ServiceLatchedCount = 1,
	Message := 'Empty hooks preserve configured and Service alarm aggregation.'
);
AssertTrue(
	Condition :=
		RegressionModule.ModuleAlarmList[1].ServiceId = 11
		AND RegressionModule.ModuleAlarmList[2].ServiceId = 0,
	Message := 'Legacy Service and JSON publication ordering is preserved.'
);
AssertTrue(
	Condition :=
		RegressionModule.ModuleStatus.Variable.PublishedCount = 1
		AND RegressionModule.ModuleVariableList[1].Id = 8001
		AND RegressionModule.ModuleVariableList[1].Value = LREAL_TO_STRING(42.0),
	Message := 'Empty hooks preserve configured SVID publication.'
);
AssertTrue(
	Condition :=
		RegressionModule.ModuleStatus.Data.PublishedCount = 1
		AND RegressionModule.ModuleDataList[1].Id = 7001
		AND RegressionModule.ModuleDataList[1].Value = '123',
	Message := 'DVID aggregation is independent of the new SVID hooks.'
);
bFinished := TRUE;

TEST_FINISHED();
END_METHOD

END_FUNCTION_BLOCK

// ---- Fakes/FB_TestableModuleBase.TcPOU
FUNCTION_BLOCK FB_TestableModuleBase EXTENDS FB_ModuleBase
VAR
	_UpperServiceCtrl : ST_ServiceCtrl;
	_EffectiveServiceCtrl : ST_ServiceCtrl;
	_UpperServiceParam : ST_TestServiceParam;
	_EffectiveServiceParam : ST_TestServiceParam;
	_ServiceStatus : ST_ServiceStatus;
END_VAR

M_UpdateModule();

METHOD PROTECTED H_RegisterServices
M_RegisterService(
	ServiceId := 1,
	AllowCompositeCall := FALSE,
	UpperCtrl := _UpperServiceCtrl,
	EffectiveCtrl := _EffectiveServiceCtrl,
	UpperParam := _UpperServiceParam,
	EffectiveParam := _EffectiveServiceParam,
	Status := _ServiceStatus);
END_METHOD

METHOD PUBLIC M_SetServiceStatus
VAR_IN_OUT CONSTANT
	Status : ST_ServiceStatus;
END_VAR
_ServiceStatus := Status;
END_METHOD

END_FUNCTION_BLOCK

// ---- Fakes/FB_TestableHookModule.TcPOU
FUNCTION_BLOCK FB_TestableHookModule EXTENDS FB_ModuleBase
VAR_INPUT
	Axis : I_Axis_BaseUnit;
	AlarmId : UDINT := 9001;
	VariableId : UDINT := 8001;
	AlarmCount : UINT := 1;
	VariableCount : UINT := 1;
	DuplicateAlarm : BOOL;
	DuplicateVariable : BOOL;
	ProbeInvalidCalls : BOOL;
END_VAR
VAR_OUTPUT
	BaseUnitScans : UDINT;
	AlarmHookScans : UDINT;
	VariableHookScans : UDINT;
	AlarmObservedScan : UDINT;
	VariableObservedScan : UDINT;
	AlarmAccepted : BOOL;
	VariableAccepted : BOOL;
	DuplicateAlarmAccepted : BOOL;
	DuplicateVariableAccepted : BOOL;
	OutsideAlarmAccepted : BOOL;
	OutsideVariableAccepted : BOOL;
	CrossAlarmAccepted : BOOL;
	CrossVariableAccepted : BOOL;
	ZeroAlarmAccepted : BOOL;
	ZeroVariableAccepted : BOOL;
END_VAR
VAR
	_UpperServiceCtrl : ST_ServiceCtrl;
	_EffectiveServiceCtrl : ST_ServiceCtrl;
	_UpperServiceParam : ST_TestServiceParam;
	_EffectiveServiceParam : ST_TestServiceParam;
	_ServiceStatus : ST_ServiceStatus;
END_VAR

IF ProbeInvalidCalls THEN
	OutsideAlarmAccepted := M_AddAlarm(
		MainErrorId := AlarmId,
		SourceErrorId := 0,
		Message := 'Axis disabled',
		Path := 'Test.Axis',
		Severity := E_Severity.Alarm
	);
	OutsideVariableAccepted := M_AddVariable(
		Id := VariableId,
		Name := 'Axis position',
		DataType := E_DescriptorType.Float_64bit,
		Unit := 'mm',
		Value := 'outside'
	);
END_IF
M_UpdateModule();

METHOD PROTECTED H_RegisterServices
M_RegisterService(
	ServiceId := 1,
	AllowCompositeCall := FALSE,
	UpperCtrl := _UpperServiceCtrl,
	EffectiveCtrl := _EffectiveServiceCtrl,
	UpperParam := _UpperServiceParam,
	EffectiveParam := _EffectiveServiceParam,
	Status := _ServiceStatus);
END_METHOD

METHOD PROTECTED H_UpdateAlarm
VAR
	nIndex : UINT;
END_VAR
AlarmHookScans := AlarmHookScans + 1;
AlarmObservedScan := BaseUnitScans;
AlarmAccepted := FALSE;
DuplicateAlarmAccepted := FALSE;
IF ProbeInvalidCalls THEN
	CrossVariableAccepted := M_AddVariable(
		Id := VariableId,
		Name := 'Axis position',
		DataType := E_DescriptorType.Float_64bit,
		Unit := 'mm',
		Value := 'wrong hook'
	);
	ZeroAlarmAccepted := M_AddAlarm(
		MainErrorId := 0,
		SourceErrorId := 0,
		Message := 'Axis disabled',
		Path := 'Test.Axis',
		Severity := E_Severity.Alarm
	);
END_IF
IF Axis = 0 THEN
	RETURN;
END_IF
IF Axis.AxisIsDisabled THEN
	FOR nIndex := 1 TO AlarmCount DO
		AlarmAccepted := M_AddAlarm(
			MainErrorId := AlarmId + UINT_TO_UDINT(nIndex) - 1,
			SourceErrorId := 0,
			Message := 'Axis disabled',
			Path := 'Test.Axis',
			Severity := E_Severity.Alarm
		);
	END_FOR
	IF DuplicateAlarm THEN
		DuplicateAlarmAccepted := M_AddAlarm(
			MainErrorId := AlarmId,
			SourceErrorId := 0,
			Message := 'Must not replace first',
			Path := 'Test.Axis',
			Severity := E_Severity.Alarm
		);
	END_IF
END_IF
END_METHOD

METHOD PROTECTED H_UpdateBaseUnit
IF Axis <> 0 THEN
	Axis.M_CyclicUpdate();
END_IF
BaseUnitScans := BaseUnitScans + 1;
END_METHOD

METHOD PROTECTED H_UpdateVariable
VAR
	nIndex : UINT;
END_VAR
VariableHookScans := VariableHookScans + 1;
VariableObservedScan := BaseUnitScans;
VariableAccepted := FALSE;
DuplicateVariableAccepted := FALSE;
IF ProbeInvalidCalls THEN
	CrossAlarmAccepted := M_AddAlarm(
		MainErrorId := AlarmId,
		SourceErrorId := 0,
		Message := 'Axis disabled',
		Path := 'Test.Axis',
		Severity := E_Severity.Alarm
	);
	ZeroVariableAccepted := M_AddVariable(
		Id := 0,
		Name := 'Axis position',
		DataType := E_DescriptorType.Float_64bit,
		Unit := 'mm',
		Value := 'zero'
	);
END_IF
IF Axis = 0 THEN
	RETURN;
END_IF
FOR nIndex := 1 TO VariableCount DO
	VariableAccepted := M_AddVariable(
		Id := VariableId + UINT_TO_UDINT(nIndex) - 1,
		Name := 'Axis position',
		DataType := E_DescriptorType.Float_64bit,
		Unit := 'mm',
		Value := LREAL_TO_STRING(Axis.AxisActualPosition)
	);
END_FOR
IF DuplicateVariable THEN
	DuplicateVariableAccepted := M_AddVariable(
		Id := VariableId,
		Name := 'Axis position',
		DataType := E_DescriptorType.Float_64bit,
		Unit := 'mm',
		Value := 'must not replace first'
	);
END_IF
END_METHOD

END_FUNCTION_BLOCK

// ---- Fakes/FB_FakeHookValueReader.TcPOU
FUNCTION_BLOCK FB_FakeHookValueReader IMPLEMENTS I_VariableNodeReader
VAR_INPUT
	Sample : LREAL;
	SampleValid : BOOL := TRUE;
END_VAR

METHOD M_ReadNode : BOOL
VAR_INPUT
	NodeHandle : UINT;
	ExpectedDataType : E_ConfigDataType;
END_VAR
VAR_IN_OUT
	Value : ST_ConfigRawValue;
END_VAR
VAR_OUTPUT
	ErrorCode : E_ConfigValueError;
END_VAR
VAR
	nSample : DINT;
END_VAR
M_ReadNode := FALSE;
MEMSET(ADR(Value), 0, SIZEOF(Value));
ErrorCode := E_ConfigValueError.InvalidNodeHandle;
IF NOT SampleValid OR (NodeHandle = 0) THEN
	RETURN;
END_IF
CASE ExpectedDataType OF
	E_ConfigDataType.Float64:
		MEMCPY(ADR(Value.Data), ADR(Sample), SIZEOF(Sample));
	E_ConfigDataType.Integer32:
		nSample := LREAL_TO_DINT(Sample);
		MEMCPY(ADR(Value.Data), ADR(nSample), SIZEOF(nSample));
	ELSE
		ErrorCode := E_ConfigValueError.NodeDataTypeMismatch;
		RETURN;
END_CASE
ErrorCode := E_ConfigValueError.None;
M_ReadNode := TRUE;
END_METHOD

END_FUNCTION_BLOCK

// ---- POUs/Test Suites/Configuration/FB_ConfigValueSnapshotReaderTests.TcPOU
FUNCTION_BLOCK FB_ConfigValueSnapshotReaderTests EXTENDS TcUnit.FB_TestSuite

DisabledInvalidAndUnavailableInputsAreNotReady();
AllSupportedTypesAreSnapshottedInConfiguredOrder();
FirstReadErrorWins();

METHOD AllSupportedTypesAreSnapshottedInConfiguredOrder
VAR_INST
	Snapshot : FB_ConfigValueSnapshotReader;
	Config : ST_ModuleRuntimeConfig;
	FakeReader : FB_FakeVariableNodeReader;
	Reader : I_VariableNodeReader;
	bValid : BOOL;
END_VAR
TEST('AllSupportedTypesAreSnapshottedInConfiguredOrder');

// Arrange：前五筆 Variable 加上一筆 Alarm，驗證兩個清單合併後仍維持順序。
Config.Enabled := TRUE;
Config.Valid := TRUE;
Config.VariableCount := 5;
Config.AlarmCount := 1;
Config.VariableBindings[1].NodeHandle := 1;
Config.VariableBindings[1].Definition.DataType := E_ConfigDataType.Boolean;
Config.VariableBindings[2].NodeHandle := 2;
Config.VariableBindings[2].Definition.DataType := E_ConfigDataType.Integer32;
Config.VariableBindings[3].NodeHandle := 3;
Config.VariableBindings[3].Definition.DataType := E_ConfigDataType.UnsignedInteger32;
Config.VariableBindings[4].NodeHandle := 4;
Config.VariableBindings[4].Definition.DataType := E_ConfigDataType.Float32;
Config.VariableBindings[5].NodeHandle := 5;
Config.VariableBindings[5].Definition.DataType := E_ConfigDataType.Float64;
Config.AlarmBindings[1].NodeHandle := 6;
Config.AlarmBindings[1].Definition.DataType := E_ConfigDataType.String80;
Reader := FakeReader;

// Act。
Snapshot(RuntimeConfig := Config, VariableNodeReader := Reader);

// Assert：數值與字串轉換都取用當輪 snapshot，而不是再次呼叫 reader。
AssertTrue(
	Condition := Snapshot.Ready AND NOT Snapshot.Error,
	Message := 'All configured reads must complete.'
);
AssertTrue(
	Condition := Snapshot.M_GetLReal(SourceIndex := 1, Valid => bValid) = 1.0 AND bValid,
	Message := 'BOOL must convert to one.'
);
AssertTrue(
	Condition := Snapshot.M_GetLReal(SourceIndex := 2, Valid => bValid) = -42.0 AND bValid,
	Message := 'DINT conversion must preserve sign.'
);
AssertTrue(
	Condition := Snapshot.M_GetLReal(SourceIndex := 3, Valid => bValid) = 42.0 AND bValid,
	Message := 'UDINT conversion must preserve value.'
);
AssertTrue(
	Condition := Snapshot.M_GetLReal(SourceIndex := 5, Valid => bValid) = 25.25 AND bValid,
	Message := 'LREAL conversion must preserve precision.'
);
AssertTrue(
	Condition := Snapshot.M_GetValueString(
		SourceIndex := 6,
		Valid => bValid
	) = 'snapshot' AND bValid,
	Message := 'Alarm source follows all Variable sources.'
);
AssertTrue(
	Condition := Snapshot.M_GetValueString(
		SourceIndex := 0,
		Valid => bValid
	) = '' AND NOT bValid,
	Message := 'Out-of-range source index must be invalid.'
);

TEST_FINISHED();
END_METHOD

METHOD DisabledInvalidAndUnavailableInputsAreNotReady
VAR_INST
	Snapshot : FB_ConfigValueSnapshotReader;
	Config : ST_ModuleRuntimeConfig;
	FakeReader : FB_FakeVariableNodeReader;
	Reader : I_VariableNodeReader;
END_VAR
TEST('DisabledInvalidAndUnavailableInputsAreNotReady');

// Arrange：disabled configuration 不應被視為錯誤，只是不 Ready。
Config.Enabled := FALSE;
Config.Valid := TRUE;
Snapshot(RuntimeConfig := Config, VariableNodeReader := Reader);
AssertFalse(
	Condition := Snapshot.Ready OR Snapshot.Error,
	Message := 'A disabled configuration must remain quietly not ready.'
);

// Act：啟用有效 config，但不提供 reader。
Config.Enabled := TRUE;
Snapshot(RuntimeConfig := Config, VariableNodeReader := Reader);
AssertTrue(
	Condition := Snapshot.Error
		AND (Snapshot.ErrorCode = E_ConfigValueError.ReaderUnavailable),
	Message := 'Missing reader must report ReaderUnavailable.'
);

// Assert：總 source 數超過固定容量時，在讀 array 前即拒絕。
Config.VariableCount := Param_Config.MaxModuleVariable;
Config.AlarmCount := Param_Config.MaxConfiguredAlarmsPerModule + 1;
Reader := FakeReader;
Snapshot(RuntimeConfig := Config, VariableNodeReader := Reader);
AssertTrue(
	Condition := Snapshot.Error
		AND (Snapshot.ErrorCode = E_ConfigValueError.SourceCapacityExceeded),
	Message := 'Source count beyond fixed capacity must be rejected before array reads.'
);

TEST_FINISHED();
END_METHOD

METHOD FirstReadErrorWins
VAR_INST
	Snapshot : FB_ConfigValueSnapshotReader;
	Config : ST_ModuleRuntimeConfig;
	FakeReader : FB_FakeVariableNodeReader;
	Reader : I_VariableNodeReader;
END_VAR
TEST('FirstReadErrorWins');

// Arrange：第二筆讀取失敗，後續來源仍可被掃描，但公開錯誤保留第一筆來源。
Config.Enabled := TRUE;
Config.Valid := TRUE;
Config.VariableCount := 3;
Config.VariableBindings[1].NodeHandle := 1;
Config.VariableBindings[1].Definition.DataType := E_ConfigDataType.Boolean;
Config.VariableBindings[1].Definition.Source := 'first';
Config.VariableBindings[2].NodeHandle := 2;
Config.VariableBindings[2].Definition.DataType := E_ConfigDataType.Integer32;
Config.VariableBindings[2].Definition.Source := 'second';
Config.VariableBindings[3].NodeHandle := 3;
Config.VariableBindings[3].Definition.DataType := E_ConfigDataType.UnsignedInteger32;
Config.VariableBindings[3].Definition.Source := 'third';
FakeReader.FailHandle := 2;
Reader := FakeReader;

Snapshot(RuntimeConfig := Config, VariableNodeReader := Reader);
AssertTrue(
	Condition := Snapshot.Error AND NOT Snapshot.Ready,
	Message := 'Any source failure must make the snapshot not ready.'
);
AssertTrue(
	Condition :=
		(Snapshot.ErrorCode = E_ConfigValueError.InvalidNodeHandle)
		AND (Snapshot.ErrorSource = 'second'),
	Message := 'The first failing source must own the diagnostic.'
);

TEST_FINISHED();
END_METHOD

END_FUNCTION_BLOCK

// ---- Fakes/FB_FakeVariableNodeReader.TcPOU
FUNCTION_BLOCK FB_FakeVariableNodeReader IMPLEMENTS I_VariableNodeReader
VAR_INPUT
	FailHandle : UINT;
END_VAR
VAR
	_BoolValue : BOOL := TRUE;
	_DIntValue : DINT := -42;
	_UDIntValue : UDINT := 42;
	_RealValue : REAL := 12.5;
	_LRealValue : LREAL := 25.25;
	_StringValue : STRING(80) := 'snapshot';
END_VAR

METHOD PUBLIC M_ReadNode : BOOL
VAR_INPUT
	NodeHandle : UINT;
	ExpectedDataType : E_ConfigDataType;
END_VAR
VAR_IN_OUT
	Value : ST_ConfigRawValue;
END_VAR
VAR_OUTPUT
	ErrorCode : E_ConfigValueError;
END_VAR
M_ReadNode := FALSE;
ErrorCode := E_ConfigValueError.None;
MEMSET(ADR(Value), 0, SIZEOF(Value));
IF NodeHandle = FailHandle THEN
	ErrorCode := E_ConfigValueError.InvalidNodeHandle;
	RETURN;
END_IF
CASE NodeHandle OF
	1:
		IF ExpectedDataType <>
			E_ConfigDataType.Boolean THEN ErrorCode := E_ConfigValueError.NodeDataTypeMismatch;
		RETURN;
		END_IF MEMCPY(ADR(Value.Data), ADR(_BoolValue), SIZEOF(_BoolValue));
	2:
		IF ExpectedDataType <>
			E_ConfigDataType.Integer32 THEN ErrorCode := E_ConfigValueError.NodeDataTypeMismatch;
		RETURN;
		END_IF MEMCPY(ADR(Value.Data), ADR(_DIntValue), SIZEOF(_DIntValue));
	3:
		IF ExpectedDataType <>
			E_ConfigDataType.UnsignedInteger32 THEN ErrorCode := E_ConfigValueError.NodeDataTypeMismatch;
		RETURN;
		END_IF MEMCPY(ADR(Value.Data), ADR(_UDIntValue), SIZEOF(_UDIntValue));
	4:
		IF ExpectedDataType <>
			E_ConfigDataType.Float32 THEN ErrorCode := E_ConfigValueError.NodeDataTypeMismatch;
		RETURN;
		END_IF MEMCPY(ADR(Value.Data), ADR(_RealValue), SIZEOF(_RealValue));
	5:
		IF ExpectedDataType <>
			E_ConfigDataType.Float64 THEN ErrorCode := E_ConfigValueError.NodeDataTypeMismatch;
		RETURN;
		END_IF MEMCPY(ADR(Value.Data), ADR(_LRealValue), SIZEOF(_LRealValue));
	6:
		IF ExpectedDataType <>
			E_ConfigDataType.String80 THEN ErrorCode := E_ConfigValueError.NodeDataTypeMismatch;
		RETURN;
		END_IF MEMCPY(ADR(Value.Data), ADR(_StringValue), SIZEOF(_StringValue));
	ELSE
		ErrorCode := E_ConfigValueError.InvalidNodeHandle;
		RETURN;
END_CASE
M_ReadNode := TRUE;
END_METHOD

END_FUNCTION_BLOCK

// ---- POUs/Test Suites/Configuration/FB_LinkVariableManagerTests.TcPOU
FUNCTION_BLOCK FB_LinkVariableManagerTests EXTENDS TcUnit.FB_TestSuite

RegistrationSessionsEnforceOrderAndRollback();
MemcpyAndNumericTransformRunOnlyInTheirPhase();
ReadableNodeAndSingleWriterValidationAreExplicit();

METHOD RegistrationSessionsEnforceOrderAndRollback
VAR_INST
	Manager : FB_LinkVariableManager;
END_VAR
VAR
	bOk : BOOL;
END_VAR
TEST('RegistrationSessionsEnforceOrderAndRollback');

// Act / Assert：session 外註冊必須失敗。
bOk := Manager.M_RegisterInfrastructureNode(
	Variable := GVL_TestSymbols.InfrastructureBool,
	Access := E_VariableAccess.ReadOnly
);
AssertFalse(
	Condition := bOk,
	Message := 'Infrastructure node requires an active session.'
);

// Begin 會清除先前錯誤；重複 Begin 產生 first-error，Seal 則 rollback 未完成內容。
AssertTrue(
	Condition := Manager.M_BeginInfrastructureRegistration(),
	Message := 'Infrastructure session must begin.'
);
AssertFalse(
	Condition := Manager.M_BeginInfrastructureRegistration(),
	Message := 'A second active infrastructure session must be rejected.'
);
AssertFalse(
	Condition := Manager.M_SealInfrastructureRegistration(),
	Message := 'Sealing a failed session must rollback.'
);

// rollback 後可以從乾淨狀態重新註冊並 seal。
AssertTrue(
	Condition := Manager.M_BeginInfrastructureRegistration(),
	Message := 'A rolled-back manager must allow a new session.'
);
AssertTrue(
	Condition := Manager.M_RegisterInfrastructureNode(
		Variable := GVL_TestSymbols.InfrastructureBool,
		Access := E_VariableAccess.ReadOnly
	),
	Message := 'Supported BOOL node must register.'
);
AssertTrue(
	Condition := Manager.M_SealInfrastructureRegistration(),
	Message := 'Valid infrastructure registration must seal.'
);

TEST_FINISHED();
END_METHOD

METHOD MemcpyAndNumericTransformRunOnlyInTheirPhase
VAR_INST
	Manager : FB_LinkVariableManager;
	Json : FB_JsonReadWriteDataType;
	ModuleConfig : ST_ModuleFileConfig;
	bInitialized : BOOL;
END_VAR
VAR
	bOk : BOOL;
	sInfraBool : STRING(255);
	sInfraLReal : STRING(255);
	sModule : STRING(255);
	sInput : STRING(255);
	sLongReal : STRING(255);
	hr : HRESULT;
END_VAR
TEST('MemcpyAndNumericTransformRunOnlyInTheirPhase');

IF NOT bInitialized THEN
	// Arrange：建立 Infrastructure 與 Module node registry。
	AssertTrue(
		Condition := Manager.M_BeginInfrastructureRegistration(),
		Message := 'Infrastructure registration must begin.'
	);
	AssertTrue(
		Condition := Manager.M_RegisterInfrastructureNode(
			Variable := GVL_TestSymbols.InfrastructureBool,
			Access := E_VariableAccess.ReadOnly
		),
		Message := 'BOOL source must register.'
	);
	AssertTrue(
		Condition := Manager.M_RegisterInfrastructureNode(
			Variable := GVL_TestSymbols.InfrastructureLReal,
			Access := E_VariableAccess.ReadOnly
		),
		Message := 'LREAL source must register.'
	);
	AssertTrue(
		Condition := Manager.M_SealInfrastructureRegistration(),
		Message := 'Infrastructure nodes must seal.'
	);
	AssertTrue(
		Condition := Manager.M_BeginModuleRegistration(
			Address := ADR(GVL_TestSymbols.ModuleOne),
			Size := SIZEOF(GVL_TestSymbols.ModuleOne),
			ModuleConfig := ModuleConfig
		),
		Message := 'Module registration must begin.'
	);
	AssertTrue(
		Condition := Manager.M_RegisterModuleNode(
			Variable := GVL_TestSymbols.ModuleOne.InputBool,
			Access := E_VariableAccess.ReadWrite
		),
		Message := 'Module BOOL target must register.'
	);
	AssertTrue(
		Condition := Manager.M_RegisterModuleNode(
			Variable := GVL_TestSymbols.ModuleOne.LongRealValue,
			Access := E_VariableAccess.ReadWrite
		),
		Message := 'Module numeric target must register.'
	);
	AssertTrue(
		Condition := Manager.M_EndModuleRegistration(ModuleSymbol => sModule),
		Message := 'Module registration must end.'
	);

